LIN {X 0,Y 573.243,Z 369.081,A -85,B 0,C 180,E1 -2301.298,E2 -2301.298} C_VEL
LIN {X 0,Y 573.218,Z 369.085,A -85,B 0,C 180,E1 -2304.019,E2 -2304.019} C_VEL
LIN {X 0,Y 573.243,Z 369.081,A -85,B 0,C 180,E1 -2306.516,E2 -2306.516} C_VEL
LIN {X 0,Y 573.233,Z 369.084,A -85,B 0,C 180,E1 -2309.118,E2 -2309.118} C_VEL
LIN {X 0,Y 573.24,Z 369.081,A -85,B 0,C 180,E1 -2311.435,E2 -2311.435} C_VEL
LIN {X 0,Y 573.267,Z 369.078,A -85,B 0,C 180,E1 -2313.81,E2 -2313.81} C_VEL
LIN {X 0,Y 573.232,Z 369.084,A -85,B 0,C 180,E1 -2316.134,E2 -2316.134} C_VEL
LIN {X 0,Y 573.254,Z 369.081,A -85,B 0,C 180,E1 -2319.174,E2 -2319.174} C_VEL
LIN {X 0,Y 573.232,Z 369.084,A -85,B 0,C 180,E1 -2321.411,E2 -2321.411} C_VEL
LIN {X 0,Y 573.253,Z 369.082,A -85,B 0,C 180,E1 -2323.622,E2 -2323.622} C_VEL
LIN {X 0,Y 573.276,Z 369.078,A -85,B 0,C 180,E1 -2325.807,E2 -2325.807} C_VEL
LIN {X 0,Y 573.267,Z 369.08,A -85,B 0,C 180,E1 -2328.745,E2 -2328.745} C_VEL
LIN {X 0,Y 573.292,Z 369.075,A -85,B 0,C 180,E1 -2331.541,E2 -2331.541} C_VEL
LIN {X 0,Y 573.291,Z 369.075,A -85,B 0,C 180,E1 -2334.372,E2 -2334.372} C_VEL
LIN {X 0,Y 573.314,Z 369.074,A -85,B 0,C 180,E1 -2337.892,E2 -2337.892} C_VEL
LIN {X 0,Y 573.331,Z 369.07,A -85,B 0,C 180,E1 -2340.702,E2 -2340.702} C_VEL
LIN {X 0,Y 573.238,Z 369.082,A -85,B 0,C 180,E1 -2343.514,E2 -2343.514} C_VEL
LIN {X 0,Y 573.294,Z 369.075,A -85,B 0,C 180,E1 -2345.628,E2 -2345.628} C_VEL
LIN {X 0,Y 573.292,Z 369.076,A -85,B 0,C 180,E1 -2348.459,E2 -2348.459} C_VEL
LIN {X 0,Y 573.275,Z 369.078,A -85,B 0,C 180,E1 -2351.312,E2 -2351.312} C_VEL
LIN {X 0,Y 573.284,Z 369.078,A -85,B 0,C 180,E1 -2354.424,E2 -2354.424} C_VEL
LIN {X 0,Y 573.262,Z 369.079,A -85,B 0,C 180,E1 -2357.111,E2 -2357.111} C_VEL
LIN {X 0,Y 573.244,Z 369.081,A -85,B 0,C 180,E1 -2360.077,E2 -2360.077} C_VEL
LIN {X 0,Y 573.237,Z 369.082,A -85,B 0,C 180,E1 -2362.338,E2 -2362.338} C_VEL
LIN {X 0,Y 573.254,Z 369.079,A -85,B 0,C 180,E1 -2364.39,E2 -2364.39} C_VEL
LIN {X 0,Y 572.627,Z 369.16,A -85,B 0,C 180,E1 -2364.976,E2 -2364.976} C_VEL
LIN {X 0,Y 569.784,Z 369.514,A -85,B 0,C 180,E1 -2365.927,E2 -2365.927} C_VEL
LIN {X 0,Y 567.352,Z 369.817,A -85,B 0,C 180,E1 -2366.693,E2 -2366.693} C_VEL
LIN {X 0,Y 566.297,Z 369.948,A -85,B 0,C 180,E1 -2367.284,E2 -2367.284} C_VEL
LIN {X 0,Y 566.207,Z 369.957,A -85,B 0,C 180,E1 -2367.484,E2 -2367.484} C_VEL
LIN {X 0,Y 566.205,Z 369.958,A -85,B 0,C 180,E1 -2369.769,E2 -2369.769} C_VEL
LIN {X 0,Y 566.208,Z 369.958,A -85,B 0,C 180,E1 -2372.43,E2 -2372.43} C_VEL
LIN {X 0,Y 566.184,Z 369.961,A -85,B 0,C 180,E1 -2374.989,E2 -2374.989} C_VEL
LIN {X 0,Y 566.2,Z 369.961,A -85,B 0,C 180,E1 -2377.461,E2 -2377.461} C_VEL
LIN {X 0,Y 566.211,Z 369.957,A -85,B 0,C 180,E1 -2380.199,E2 -2380.199} C_VEL
LIN {X 0,Y 566.204,Z 369.958,A -85,B 0,C 180,E1 -2383.054,E2 -2383.054} C_VEL
LIN {X 0,Y 566.198,Z 369.958,A -85,B 0,C 180,E1 -2386.049,E2 -2386.049} C_VEL
LIN {X 0,Y 566.185,Z 369.963,A -85,B 0,C 180,E1 -2388.861,E2 -2388.861} C_VEL
LIN {X 0,Y 566.218,Z 369.956,A -85,B 0,C 180,E1 -2391.441,E2 -2391.441} C_VEL
LIN {X 0,Y 566.168,Z 369.963,A -85,B 0,C 180,E1 -2394.307,E2 -2394.307} C_VEL
LIN {X 0,Y 566.225,Z 369.957,A -85,B 0,C 180,E1 -2396.897,E2 -2396.897} C_VEL
LIN {X 0,Y 566.181,Z 369.961,A -85,B 0,C 180,E1 -2399.406,E2 -2399.406} C_VEL
LIN {X 0,Y 566.2,Z 369.958,A -85,B 0,C 180,E1 -2401.856,E2 -2401.856} C_VEL
LIN {X 0,Y 566.219,Z 369.957,A -85,B 0,C 180,E1 -2404.25,E2 -2404.25} C_VEL
LIN {X 0,Y 566.178,Z 369.962,A -85,B 0,C 180,E1 -2406.718,E2 -2406.718} C_VEL
LIN {X 0,Y 566.219,Z 369.957,A -85,B 0,C 180,E1 -2409.662,E2 -2409.662} C_VEL
LIN {X 0,Y 566.205,Z 369.96,A -85,B 0,C 180,E1 -2412.667,E2 -2412.667} C_VEL
LIN {X 0,Y 566.24,Z 369.955,A -85,B 0,C 180,E1 -2415.626,E2 -2415.626} C_VEL
LIN {X 0,Y 566.111,Z 369.972,A -85,B 0,C 180,E1 -2418.542,E2 -2418.542} C_VEL
LIN {X 0,Y 566.05,Z 370.2,A -85,B 0,C 180,E1 -2419.266,E2 -2419.266} C_VEL
LIN {X 0,Y 566.031,Z 373.545,A -85,B 0,C 180,E1 -2422.149,E2 -2422.149} C_VEL
LIN {X 0,Y 566.036,Z 376.76,A -85,B 0,C 180,E1 -2425.013,E2 -2425.013} C_VEL
LIN {X 0,Y 565.932,Z 379.928,A -85,B 0,C 180,E1 -2427.864,E2 -2427.864} C_VEL
LIN {X 0,Y 565.858,Z 383.215,A -85,B 0,C 180,E1 -2430.71,E2 -2430.71} C_VEL
LIN {X 0,Y 565.899,Z 386.764,A -85,B 0,C 180,E1 -2433.559,E2 -2433.559} C_VEL
LIN {X 0,Y 565.875,Z 390.539,A -85,B 0,C 180,E1 -2436.497,E2 -2436.497} C_VEL
LIN {X 0,Y 565.805,Z 394.183,A -85,B 0,C 180,E1 -2439.291,E2 -2439.291} C_VEL
LIN {X 0,Y 565.863,Z 395.844,A -85,B 0,C 180,E1 -2440.441,E2 -2440.441} C_VEL
LIN {X 0,Y 566.862,Z 403.182,A -85,B 0,C 180,E1 -2440.626,E2 -2440.626} C_VEL
LIN {X 0,Y 566.816,Z 416.303,A -85,B 0,C 180,E1 -2441.032,E2 -2441.032} C_VEL
LIN {X 0,Y 566.624,Z 427.611,A -85,B 0,C 180,E1 -2441.518,E2 -2441.518} C_VEL
LIN {X 0,Y 566.478,Z 439.306,A -85,B 0,C 180,E1 -2442.174,E2 -2442.174} C_VEL
LIN {X 0,Y 566.351,Z 450.857,A -85,B 0,C 180,E1 -2442.996,E2 -2442.996} C_VEL
LIN {X 0,Y 566.205,Z 460.179,A -85,B 0,C 180,E1 -2443.822,E2 -2443.822} C_VEL
LIN {X 0,Y 566.12,Z 468.385,A -85,B 0,C 180,E1 -2444.705,E2 -2444.705} C_VEL
LIN {X 0,Y 566.031,Z 477.042,A -85,B 0,C 180,E1 -2445.851,E2 -2445.851} C_VEL
LIN {X 0,Y 565.988,Z 484.113,A -85,B 0,C 180,E1 -2447.035,E2 -2447.035} C_VEL
LIN {X 0,Y 565.927,Z 489.058,A -85,B 0,C 180,E1 -2448.085,E2 -2448.085} C_VEL
LIN {X 0,Y 565.888,Z 493.37,A -85,B 0,C 180,E1 -2449.287,E2 -2449.287} C_VEL
LIN {X 0,Y 565.86,Z 496.126,A -85,B 0,C 180,E1 -2450.349,E2 -2450.349} C_VEL
LIN {X 0,Y 565.859,Z 497.849,A -85,B 0,C 180,E1 -2451.329,E2 -2451.329} C_VEL
LIN {X 0,Y 565.839,Z 498.918,A -85,B 0,C 180,E1 -2452.644,E2 -2452.644} C_VEL
LIN {X 0,Y 565.845,Z 498.924,A -85,B 0,C 180,E1 -2453.417,E2 -2453.417} C_VEL
LIN {X 0,Y 565.826,Z 498.482,A -85,B 0,C 180,E1 -2454.196,E2 -2454.196} C_VEL
LIN {X 0,Y 565.847,Z 497.517,A -85,B 0,C 180,E1 -2454.977,E2 -2454.977} C_VEL
LIN {X 0,Y 565.853,Z 496.078,A -85,B 0,C 180,E1 -2455.765,E2 -2455.765} C_VEL
LIN {X 0,Y 565.901,Z 492.922,A -85,B 0,C 180,E1 -2456.953,E2 -2456.953} C_VEL
LIN {X 0,Y 565.923,Z 488.418,A -85,B 0,C 180,E1 -2458.156,E2 -2458.156} C_VEL
LIN {X 0,Y 565.975,Z 482.771,A -85,B 0,C 180,E1 -2459.301,E2 -2459.301} C_VEL
LIN {X 0,Y 566.088,Z 476.006,A -85,B 0,C 180,E1 -2460.39,E2 -2460.39} C_VEL
LIN {X 0,Y 566.15,Z 468.073,A -85,B 0,C 180,E1 -2461.422,E2 -2461.422} C_VEL
LIN {X 0,Y 566.279,Z 458.336,A -85,B 0,C 180,E1 -2462.442,E2 -2462.442} C_VEL
LIN {X 0,Y 566.385,Z 448.167,A -85,B 0,C 180,E1 -2463.301,E2 -2463.301} C_VEL
LIN {X 0,Y 566.54,Z 437.358,A -85,B 0,C 180,E1 -2464.038,E2 -2464.038} C_VEL
LIN {X 0,Y 566.692,Z 425.446,A -85,B 0,C 180,E1 -2464.673,E2 -2464.673} C_VEL
LIN {X 0,Y 566.777,Z 412.677,A -85,B 0,C 180,E1 -2465.186,E2 -2465.186} C_VEL
LIN {X 0,Y 566.713,Z 400.738,A -85,B 0,C 180,E1 -2465.528,E2 -2465.528} C_VEL
LIN {X 0,Y 565.86,Z 395.663,A -85,B 0,C 180,E1 -2465.673,E2 -2465.673} C_VEL
LIN {X 0,Y 565.839,Z 391.945,A -85,B 0,C 180,E1 -2468.511,E2 -2468.511} C_VEL
LIN {X 0,Y 565.879,Z 388.515,A -85,B 0,C 180,E1 -2471.163,E2 -2471.163} C_VEL
LIN {X 0,Y 565.888,Z 384.824,A -85,B 0,C 180,E1 -2474.063,E2 -2474.063} C_VEL
LIN {X 0,Y 565.914,Z 382.456,A -85,B 0,C 180,E1 -2476.075,E2 -2476.075} C_VEL
LIN {X 0,Y 565.949,Z 379.413,A -85,B 0,C 180,E1 -2478.84,E2 -2478.84} C_VEL
LIN {X 0,Y 565.95,Z 376.333,A -85,B 0,C 180,E1 -2481.618,E2 -2481.618} C_VEL
LIN {X 0,Y 566.006,Z 373.303,A -85,B 0,C 180,E1 -2484.296,E2 -2484.296} C_VEL
LIN {X 0,Y 566.029,Z 370.291,A -85,B 0,C 180,E1 -2486.885,E2 -2486.885} C_VEL
LIN {X 0,Y 566.128,Z 369.968,A -85,B 0,C 180,E1 -2488.574,E2 -2488.574} C_VEL
LIN {X 0,Y 566.181,Z 369.963,A -85,B 0,C 180,E1 -2491.046,E2 -2491.046} C_VEL
LIN {X 0,Y 566.229,Z 369.955,A -85,B 0,C 180,E1 -2493.46,E2 -2493.46} C_VEL
LIN {X 0,Y 566.198,Z 369.957,A -85,B 0,C 180,E1 -2495.819,E2 -2495.819} C_VEL
LIN {X 0,Y 566.196,Z 369.957,A -85,B 0,C 180,E1 -2498.576,E2 -2498.576} C_VEL
LIN {X 0,Y 566.202,Z 369.956,A -85,B 0,C 180,E1 -2501.172,E2 -2501.172} C_VEL
LIN {X 0,Y 566.19,Z 369.958,A -85,B 0,C 180,E1 -2504.152,E2 -2504.152} C_VEL
LIN {X 0,Y 566.186,Z 369.958,A -85,B 0,C 180,E1 -2506.359,E2 -2506.359} C_VEL
LIN {X 0,Y 566.235,Z 369.952,A -85,B 0,C 180,E1 -2509.27,E2 -2509.27} C_VEL
LIN {X 0,Y 566.226,Z 369.954,A -85,B 0,C 180,E1 -2512.153,E2 -2512.153} C_VEL
LIN {X 0,Y 566.274,Z 369.949,A -85,B 0,C 180,E1 -2515.016,E2 -2515.016} C_VEL
LIN {X 0,Y 566.275,Z 369.95,A -85,B 0,C 180,E1 -2517.866,E2 -2517.866} C_VEL
LIN {X 0,Y 566.293,Z 369.949,A -85,B 0,C 180,E1 -2520.711,E2 -2520.711} C_VEL
LIN {X 0,Y 566.264,Z 369.948,A -85,B 0,C 180,E1 -2522.846,E2 -2522.846} C_VEL
LIN {X 0,Y 566.244,Z 369.951,A -85,B 0,C 180,E1 -2525.699,E2 -2525.699} C_VEL
LIN {X 0,Y 566.214,Z 369.956,A -85,B 0,C 180,E1 -2528.566,E2 -2528.566} C_VEL
LIN {X 0,Y 566.23,Z 369.956,A -85,B 0,C 180,E1 -2531.455,E2 -2531.455} C_VEL
LIN {X 0,Y 566.213,Z 369.957,A -85,B 0,C 180,E1 -2534.508,E2 -2534.508} C_VEL
LIN {X 0,Y 566.186,Z 369.96,A -85,B 0,C 180,E1 -2537.332,E2 -2537.332} C_VEL
LIN {X 0,Y 566.197,Z 369.96,A -85,B 0,C 180,E1 -2539.581,E2 -2539.581} C_VEL
LIN {X 0,Y 566.207,Z 369.958,A -85,B 0,C 180,E1 -2542.631,E2 -2542.631} C_VEL
LIN {X 0,Y 566.198,Z 369.961,A -85,B 0,C 180,E1 -2545.031,E2 -2545.031} C_VEL
LIN {X 0,Y 566.209,Z 369.957,A -85,B 0,C 180,E1 -2547.339,E2 -2547.339} C_VEL
LIN {X 0,Y 566.185,Z 369.959,A -85,B 0,C 180,E1 -2549.77,E2 -2549.77} C_VEL
LIN {X 0,Y 566.194,Z 369.958,A -85,B 0,C 180,E1 -2552.433,E2 -2552.433} C_VEL
LIN {X 0,Y 566.198,Z 369.958,A -85,B 0,C 180,E1 -2554.996,E2 -2554.996} C_VEL
LIN {X 0,Y 566.182,Z 369.962,A -85,B 0,C 180,E1 -2557.462,E2 -2557.462} C_VEL
LIN {X 0,Y 566.211,Z 369.958,A -85,B 0,C 180,E1 -2560.199,E2 -2560.199} C_VEL
LIN {X 0,Y 566.188,Z 369.961,A -85,B 0,C 180,E1 -2563.056,E2 -2563.056} C_VEL
LIN {X 0,Y 566.19,Z 369.96,A -85,B 0,C 180,E1 -2566.05,E2 -2566.05} C_VEL
LIN {X 0,Y 566.21,Z 369.957,A -85,B 0,C 180,E1 -2568.866,E2 -2568.866} C_VEL
LIN {X 0,Y 566.18,Z 369.961,A -85,B 0,C 180,E1 -2571.639,E2 -2571.639} C_VEL
LIN {X 0,Y 566.233,Z 370.124,A -85,B 0,C 180,E1 -2573.047,E2 -2573.047} C_VEL
LIN {X 0,Y 566.84,Z 373.924,A -85,B 0,C 180,E1 -2574.36,E2 -2574.36} C_VEL
LIN {X 0,Y 566.738,Z 381.867,A -85,B 0,C 180,E1 -2576.934,E2 -2576.934} C_VEL
LIN {X 0,Y 566.604,Z 389.811,A -85,B 0,C 180,E1 -2579.435,E2 -2579.435} C_VEL
LIN {X 0,Y 566.501,Z 399.078,A -85,B 0,C 180,E1 -2582.277,E2 -2582.277} C_VEL
LIN {X 0,Y 566.407,Z 408.345,A -85,B 0,C 180,E1 -2585.049,E2 -2585.049} C_VEL
LIN {X 0,Y 566.319,Z 418.936,A -85,B 0,C 180,E1 -2588.144,E2 -2588.144} C_VEL
LIN {X 0,Y 566.19,Z 429.527,A -85,B 0,C 180,E1 -2591.174,E2 -2591.174} C_VEL
LIN {X 0,Y 566.114,Z 440.118,A -85,B 0,C 180,E1 -2594.152,E2 -2594.152} C_VEL
LIN {X 0,Y 566.022,Z 449.385,A -85,B 0,C 180,E1 -2596.722,E2 -2596.722} C_VEL
LIN {X 0,Y 566.013,Z 451.536,A -85,B 0,C 180,E1 -2597.315,E2 -2597.315} C_VEL
LIN {X 0,Y 566.93,Z 458.454,A -85,B 0,C 180,E1 -2597.472,E2 -2597.472} C_VEL
LIN {X 0,Y 566.856,Z 470.552,A -85,B 0,C 180,E1 -2597.789,E2 -2597.789} C_VEL
LIN {X 0,Y 566.69,Z 482.355,A -85,B 0,C 180,E1 -2598.23,E2 -2598.23} C_VEL
LIN {X 0,Y 566.541,Z 494.944,A -85,B 0,C 180,E1 -2598.866,E2 -2598.866} C_VEL
LIN {X 0,Y 566.432,Z 505.501,A -85,B 0,C 180,E1 -2599.547,E2 -2599.547} C_VEL
LIN {X 0,Y 566.3,Z 515.665,A -85,B 0,C 180,E1 -2600.357,E2 -2600.357} C_VEL
LIN {X 0,Y 566.165,Z 524.801,A -85,B 0,C 180,E1 -2601.255,E2 -2601.255} C_VEL
LIN {X 0,Y 566.079,Z 533.702,A -85,B 0,C 180,E1 -2602.332,E2 -2602.332} C_VEL
LIN {X 0,Y 565.966,Z 540.964,A -85,B 0,C 180,E1 -2603.424,E2 -2603.424} C_VEL
LIN {X 0,Y 566.003,Z 545.688,A -85,B 0,C 180,E1 -2604.301,E2 -2604.301} C_VEL
LIN {X 0,Y 565.933,Z 550.377,A -85,B 0,C 180,E1 -2605.372,E2 -2605.372} C_VEL
LIN {X 0,Y 565.926,Z 553.961,A -85,B 0,C 180,E1 -2606.441,E2 -2606.441} C_VEL
LIN {X 0,Y 565.877,Z 555.812,A -85,B 0,C 180,E1 -2607.154,E2 -2607.154} C_VEL
LIN {X 0,Y 565.84,Z 557.202,A -85,B 0,C 180,E1 -2607.866,E2 -2607.866} C_VEL
LIN {X 0,Y 565.841,Z 558.785,A -85,B 0,C 180,E1 -2609.29,E2 -2609.29} C_VEL
LIN {X 0,Y 565.839,Z 559,A -85,B 0,C 180,E1 -2610.001,E2 -2610.001} C_VEL
LIN {X 0,Y 565.846,Z 558.184,A -85,B 0,C 180,E1 -2611.425,E2 -2611.425} C_VEL
LIN {X 0,Y 565.841,Z 557.199,A -85,B 0,C 180,E1 -2612.137,E2 -2612.137} C_VEL
LIN {X 0,Y 565.878,Z 555.807,A -85,B 0,C 180,E1 -2612.849,E2 -2612.849} C_VEL
LIN {X 0,Y 565.927,Z 552.892,A -85,B 0,C 180,E1 -2613.918,E2 -2613.918} C_VEL
LIN {X 0,Y 565.878,Z 548.944,A -85,B 0,C 180,E1 -2614.989,E2 -2614.989} C_VEL
LIN {X 0,Y 566.002,Z 543.86,A -85,B 0,C 180,E1 -2616.06,E2 -2616.06} C_VEL
LIN {X 0,Y 566.042,Z 537.461,A -85,B 0,C 180,E1 -2617.134,E2 -2617.134} C_VEL
LIN {X 0,Y 566.134,Z 529.468,A -85,B 0,C 180,E1 -2618.209,E2 -2618.209} C_VEL
LIN {X 0,Y 566.23,Z 521.325,A -85,B 0,C 180,E1 -2619.107,E2 -2619.107} C_VEL
LIN {X 0,Y 566.347,Z 511.388,A -85,B 0,C 180,E1 -2620.006,E2 -2620.006} C_VEL
LIN {X 0,Y 566.52,Z 500.298,A -85,B 0,C 180,E1 -2620.807,E2 -2620.807} C_VEL
LIN {X 0,Y 566.611,Z 487.929,A -85,B 0,C 180,E1 -2621.511,E2 -2621.511} C_VEL
LIN {X 0,Y 566.778,Z 475.734,A -85,B 0,C 180,E1 -2622.034,E2 -2622.034} C_VEL
LIN {X 0,Y 566.928,Z 462.304,A -85,B 0,C 180,E1 -2622.44,E2 -2622.44} C_VEL
LIN {X 0,Y 566.631,Z 455.461,A -85,B 0,C 180,E1 -2622.594,E2 -2622.594} C_VEL
LIN {X 0,Y 566.015,Z 451.526,A -85,B 0,C 180,E1 -2622.688,E2 -2622.688} C_VEL
LIN {X 0,Y 566.09,Z 441.432,A -85,B 0,C 180,E1 -2625.482,E2 -2625.482} C_VEL
LIN {X 0,Y 566.176,Z 430.841,A -85,B 0,C 180,E1 -2628.454,E2 -2628.454} C_VEL
LIN {X 0,Y 566.242,Z 421.573,A -85,B 0,C 180,E1 -2631.097,E2 -2631.097} C_VEL
LIN {X 0,Y 566.344,Z 412.306,A -85,B 0,C 180,E1 -2633.786,E2 -2633.786} C_VEL
LIN {X 0,Y 566.482,Z 403.039,A -85,B 0,C 180,E1 -2636.529,E2 -2636.529} C_VEL
LIN {X 0,Y 566.54,Z 393.772,A -85,B 0,C 180,E1 -2639.342,E2 -2639.342} C_VEL
LIN {X 0,Y 566.756,Z 384.505,A -85,B 0,C 180,E1 -2642.224,E2 -2642.224} C_VEL
LIN {X 0,Y 566.841,Z 376.562,A -85,B 0,C 180,E1 -2644.774,E2 -2644.774} C_VEL
LIN {X 0,Y 566.583,Z 372.063,A -85,B 0,C 180,E1 -2646.266,E2 -2646.266} C_VEL
LIN {X 0,Y 566.24,Z 369.954,A -85,B 0,C 180,E1 -2647.012,E2 -2647.012} C_VEL
LIN {X 0,Y 566.219,Z 369.957,A -85,B 0,C 180,E1 -2649.686,E2 -2649.686} C_VEL
LIN {X 0,Y 566.206,Z 369.958,A -85,B 0,C 180,E1 -2652.917,E2 -2652.917} C_VEL
LIN {X 0,Y 566.199,Z 369.959,A -85,B 0,C 180,E1 -2656.05,E2 -2656.05} C_VEL
LIN {X 0,Y 566.209,Z 369.958,A -85,B 0,C 180,E1 -2659.215,E2 -2659.215} C_VEL
LIN {X 0,Y 566.188,Z 369.962,A -85,B 0,C 180,E1 -2661.637,E2 -2661.637} C_VEL
LIN {X 0,Y 566.167,Z 369.963,A -85,B 0,C 180,E1 -2664.308,E2 -2664.308} C_VEL
LIN {X 0,Y 566.208,Z 369.96,A -85,B 0,C 180,E1 -2666.897,E2 -2666.897} C_VEL
LIN {X 0,Y 566.185,Z 369.96,A -85,B 0,C 180,E1 -2669.407,E2 -2669.407} C_VEL
LIN {X 0,Y 566.199,Z 369.959,A -85,B 0,C 180,E1 -2671.857,E2 -2671.857} C_VEL
LIN {X 0,Y 566.217,Z 369.959,A -85,B 0,C 180,E1 -2674.251,E2 -2674.251} C_VEL
LIN {X 0,Y 566.176,Z 369.962,A -85,B 0,C 180,E1 -2676.719,E2 -2676.719} C_VEL
LIN {X 0,Y 566.217,Z 369.957,A -85,B 0,C 180,E1 -2679.663,E2 -2679.663} C_VEL
LIN {X 0,Y 566.204,Z 369.959,A -85,B 0,C 180,E1 -2682.668,E2 -2682.668} C_VEL
LIN {X 0,Y 566.237,Z 369.956,A -85,B 0,C 180,E1 -2685.627,E2 -2685.627} C_VEL
LIN {X 0,Y 566.239,Z 369.956,A -85,B 0,C 180,E1 -2688.675,E2 -2688.675} C_VEL
LIN {X 0,Y 566.236,Z 369.953,A -85,B 0,C 180,E1 -2691.434,E2 -2691.434} C_VEL
LIN {X 0,Y 566.26,Z 369.951,A -85,B 0,C 180,E1 -2694.302,E2 -2694.302} C_VEL
LIN {X 0,Y 566.285,Z 369.949,A -85,B 0,C 180,E1 -2697.866,E2 -2697.866} C_VEL
LIN {X 0,Y 566.302,Z 369.946,A -85,B 0,C 180,E1 -2700.711,E2 -2700.711} C_VEL
LIN {X 0,Y 566.275,Z 369.949,A -85,B 0,C 180,E1 -2702.845,E2 -2702.845} C_VEL
LIN {X 0,Y 566.262,Z 369.951,A -85,B 0,C 180,E1 -2705.698,E2 -2705.698} C_VEL
LIN {X 0,Y 566.236,Z 369.954,A -85,B 0,C 180,E1 -2708.566,E2 -2708.566} C_VEL
LIN {X 0,Y 566.246,Z 369.955,A -85,B 0,C 180,E1 -2711.454,E2 -2711.454} C_VEL
LIN {X 0,Y 566.237,Z 369.956,A -85,B 0,C 180,E1 -2714.506,E2 -2714.506} C_VEL
LIN {X 0,Y 566.202,Z 369.958,A -85,B 0,C 180,E1 -2717.332,E2 -2717.332} C_VEL
LIN {X 0,Y 566.21,Z 369.957,A -85,B 0,C 180,E1 -2720.337,E2 -2720.337} C_VEL
LIN {X 0,Y 566.177,Z 369.962,A -85,B 0,C 180,E1 -2723.282,E2 -2723.282} C_VEL
LIN {X 0,Y 566.213,Z 369.958,A -85,B 0,C 180,E1 -2725.749,E2 -2725.749} C_VEL
LIN {X 0,Y 566.207,Z 369.957,A -85,B 0,C 180,E1 -2727.484,E2 -2727.484} C_VEL
LIN {X 0,Y 565.527,Z 370.044,A -85,B 0,C 180,E1 -2728.078,E2 -2728.078} C_VEL
LIN {X 0,Y 562.661,Z 370.401,A -85,B 0,C 180,E1 -2729.042,E2 -2729.042} C_VEL
LIN {X 0,Y 560.251,Z 370.7,A -85,B 0,C 180,E1 -2729.817,E2 -2729.817} C_VEL
LIN {X 0,Y 559.224,Z 370.828,A -85,B 0,C 180,E1 -2730.416,E2 -2730.416} C_VEL
LIN {X 0,Y 559.144,Z 370.837,A -85,B 0,C 180,E1 -2730.619,E2 -2730.619} C_VEL
LIN {X 0,Y 559.163,Z 370.836,A -85,B 0,C 180,E1 -2733.575,E2 -2733.575} C_VEL
LIN {X 0,Y 559.15,Z 370.838,A -85,B 0,C 180,E1 -2736.445,E2 -2736.445} C_VEL
LIN {X 0,Y 559.176,Z 370.833,A -85,B 0,C 180,E1 -2738.934,E2 -2738.934} C_VEL
LIN {X 0,Y 559.166,Z 370.835,A -85,B 0,C 180,E1 -2741.77,E2 -2741.77} C_VEL
LIN {X 0,Y 559.136,Z 370.84,A -85,B 0,C 180,E1 -2744.74,E2 -2744.74} C_VEL
LIN {X 0,Y 559.179,Z 370.834,A -85,B 0,C 180,E1 -2747.863,E2 -2747.863} C_VEL
LIN {X 0,Y 559.182,Z 370.834,A -85,B 0,C 180,E1 -2751.066,E2 -2751.066} C_VEL
LIN {X 0,Y 559.145,Z 370.839,A -85,B 0,C 180,E1 -2753.789,E2 -2753.789} C_VEL
LIN {X 0,Y 559.168,Z 370.835,A -85,B 0,C 180,E1 -2756.425,E2 -2756.425} C_VEL
LIN {X 0,Y 559.158,Z 370.837,A -85,B 0,C 180,E1 -2758.98,E2 -2758.98} C_VEL
LIN {X 0,Y 559.174,Z 370.833,A -85,B 0,C 180,E1 -2761.618,E2 -2761.618} C_VEL
LIN {X 0,Y 559.185,Z 370.831,A -85,B 0,C 180,E1 -2763.902,E2 -2763.902} C_VEL
LIN {X 0,Y 559.147,Z 370.839,A -85,B 0,C 180,E1 -2766.57,E2 -2766.57} C_VEL
LIN {X 0,Y 559.185,Z 370.834,A -85,B 0,C 180,E1 -2769.395,E2 -2769.395} C_VEL
LIN {X 0,Y 559.148,Z 370.838,A -85,B 0,C 180,E1 -2771.685,E2 -2771.685} C_VEL
LIN {X 0,Y 559.169,Z 370.835,A -85,B 0,C 180,E1 -2773.947,E2 -2773.947} C_VEL
LIN {X 0,Y 559.179,Z 370.833,A -85,B 0,C 180,E1 -2776.183,E2 -2776.183} C_VEL
LIN {X 0,Y 559.086,Z 370.847,A -85,B 0,C 180,E1 -2778.667,E2 -2778.667} C_VEL
LIN {X 0,Y 558.996,Z 370.858,A -85,B 0,C 180,E1 -2779.128,E2 -2779.128} C_VEL
LIN {X 0,Y 558.961,Z 374.055,A -85,B 0,C 180,E1 -2782.049,E2 -2782.049} C_VEL
LIN {X 0,Y 558.985,Z 377.336,A -85,B 0,C 180,E1 -2784.95,E2 -2784.95} C_VEL
LIN {X 0,Y 558.859,Z 380.549,A -85,B 0,C 180,E1 -2787.837,E2 -2787.837} C_VEL
LIN {X 0,Y 558.88,Z 382.996,A -85,B 0,C 180,E1 -2789.999,E2 -2789.999} C_VEL
LIN {X 0,Y 558.762,Z 386.292,A -85,B 0,C 180,E1 -2792.882,E2 -2792.882} C_VEL
LIN {X 0,Y 558.822,Z 389.89,A -85,B 0,C 180,E1 -2795.773,E2 -2795.773} C_VEL
LIN {X 0,Y 558.755,Z 393.622,A -85,B 0,C 180,E1 -2798.68,E2 -2798.68} C_VEL
LIN {X 0,Y 558.758,Z 395.823,A -85,B 0,C 180,E1 -2800.278,E2 -2800.278} C_VEL
LIN {X 0,Y 559.933,Z 403.771,A -85,B 0,C 180,E1 -2800.484,E2 -2800.484} C_VEL
LIN {X 0,Y 559.87,Z 416.607,A -85,B 0,C 180,E1 -2800.893,E2 -2800.893} C_VEL
LIN {X 0,Y 559.641,Z 428.895,A -85,B 0,C 180,E1 -2801.439,E2 -2801.439} C_VEL
LIN {X 0,Y 559.462,Z 440.992,A -85,B 0,C 180,E1 -2802.145,E2 -2802.145} C_VEL
LIN {X 0,Y 559.323,Z 451.065,A -85,B 0,C 180,E1 -2802.885,E2 -2802.885} C_VEL
LIN {X 0,Y 559.161,Z 461.247,A -85,B 0,C 180,E1 -2803.814,E2 -2803.814} C_VEL
LIN {X 0,Y 559.049,Z 469.59,A -85,B 0,C 180,E1 -2804.746,E2 -2804.746} C_VEL
LIN {X 0,Y 558.956,Z 477.784,A -85,B 0,C 180,E1 -2805.869,E2 -2805.869} C_VEL
LIN {X 0,Y 558.923,Z 483.323,A -85,B 0,C 180,E1 -2806.809,E2 -2806.809} C_VEL
LIN {X 0,Y 558.836,Z 488.743,A -85,B 0,C 180,E1 -2807.944,E2 -2807.944} C_VEL
LIN {X 0,Y 558.81,Z 492.914,A -85,B 0,C 180,E1 -2809.085,E2 -2809.085} C_VEL
LIN {X 0,Y 558.76,Z 495.051,A -85,B 0,C 180,E1 -2809.851,E2 -2809.851} C_VEL
LIN {X 0,Y 558.759,Z 496.735,A -85,B 0,C 180,E1 -2810.619,E2 -2810.619} C_VEL
LIN {X 0,Y 558.764,Z 498.012,A -85,B 0,C 180,E1 -2811.447,E2 -2811.447} C_VEL
LIN {X 0,Y 558.737,Z 498.683,A -85,B 0,C 180,E1 -2812.168,E2 -2812.168} C_VEL
LIN {X 0,Y 558.755,Z 498.943,A -85,B 0,C 180,E1 -2813.337,E2 -2813.337} C_VEL
LIN {X 0,Y 558.757,Z 498.145,A -85,B 0,C 180,E1 -2814.522,E2 -2814.522} C_VEL
LIN {X 0,Y 558.751,Z 497.025,A -85,B 0,C 180,E1 -2815.317,E2 -2815.317} C_VEL
LIN {X 0,Y 558.813,Z 493.652,A -85,B 0,C 180,E1 -2816.754,E2 -2816.754} C_VEL
LIN {X 0,Y 558.838,Z 489.228,A -85,B 0,C 180,E1 -2818.025,E2 -2818.025} C_VEL
LIN {X 0,Y 558.909,Z 482.859,A -85,B 0,C 180,E1 -2819.365,E2 -2819.365} C_VEL
LIN {X 0,Y 559.016,Z 475.168,A -85,B 0,C 180,E1 -2820.606,E2 -2820.606} C_VEL
LIN {X 0,Y 559.102,Z 466.635,A -85,B 0,C 180,E1 -2821.696,E2 -2821.696} C_VEL
LIN {X 0,Y 559.273,Z 456.793,A -85,B 0,C 180,E1 -2822.705,E2 -2822.705} C_VEL
LIN {X 0,Y 559.433,Z 446.565,A -85,B 0,C 180,E1 -2823.554,E2 -2823.554} C_VEL
LIN {X 0,Y 559.57,Z 435.653,A -85,B 0,C 180,E1 -2824.278,E2 -2824.278} C_VEL
LIN {X 0,Y 559.759,Z 423.899,A -85,B 0,C 180,E1 -2824.891,E2 -2824.891} C_VEL
LIN {X 0,Y 559.885,Z 410.658,A -85,B 0,C 180,E1 -2825.407,E2 -2825.407} C_VEL
LIN {X 0,Y 559.735,Z 401.403,A -85,B 0,C 180,E1 -2825.67,E2 -2825.67} C_VEL
LIN {X 0,Y 558.754,Z 395.676,A -85,B 0,C 180,E1 -2825.826,E2 -2825.826} C_VEL
LIN {X 0,Y 558.742,Z 391.618,A -85,B 0,C 180,E1 -2828.967,E2 -2828.967} C_VEL
LIN {X 0,Y 558.789,Z 388.008,A -85,B 0,C 180,E1 -2831.802,E2 -2831.802} C_VEL
LIN {X 0,Y 558.857,Z 384.581,A -85,B 0,C 180,E1 -2834.765,E2 -2834.765} C_VEL
LIN {X 0,Y 558.858,Z 381.052,A -85,B 0,C 180,E1 -2837.895,E2 -2837.895} C_VEL
LIN {X 0,Y 558.885,Z 378.677,A -85,B 0,C 180,E1 -2840.109,E2 -2840.109} C_VEL
LIN {X 0,Y 558.917,Z 375.56,A -85,B 0,C 180,E1 -2842.874,E2 -2842.874} C_VEL
LIN {X 0,Y 558.945,Z 372.481,A -85,B 0,C 180,E1 -2845.541,E2 -2845.541} C_VEL
LIN {X 0,Y 559.003,Z 370.858,A -85,B 0,C 180,E1 -2847.385,E2 -2847.385} C_VEL
LIN {X 0,Y 559.171,Z 370.833,A -85,B 0,C 180,E1 -2850.134,E2 -2850.134} C_VEL
LIN {X 0,Y 559.165,Z 370.833,A -85,B 0,C 180,E1 -2853.169,E2 -2853.169} C_VEL
LIN {X 0,Y 559.148,Z 370.836,A -85,B 0,C 180,E1 -2855.494,E2 -2855.494} C_VEL
LIN {X 0,Y 559.146,Z 370.835,A -85,B 0,C 180,E1 -2858.446,E2 -2858.446} C_VEL
LIN {X 0,Y 559.156,Z 370.835,A -85,B 0,C 180,E1 -2860.926,E2 -2860.926} C_VEL
LIN {X 0,Y 559.152,Z 370.834,A -85,B 0,C 180,E1 -2863.947,E2 -2863.947} C_VEL
LIN {X 0,Y 559.16,Z 370.835,A -85,B 0,C 180,E1 -2866.184,E2 -2866.184} C_VEL
LIN {X 0,Y 559.196,Z 370.829,A -85,B 0,C 180,E1 -2869.134,E2 -2869.134} C_VEL
LIN {X 0,Y 559.194,Z 370.829,A -85,B 0,C 180,E1 -2872.054,E2 -2872.054} C_VEL
LIN {X 0,Y 559.247,Z 370.823,A -85,B 0,C 180,E1 -2874.953,E2 -2874.953} C_VEL
LIN {X 0,Y 559.244,Z 370.825,A -85,B 0,C 180,E1 -2877.839,E2 -2877.839} C_VEL
LIN {X 0,Y 559.262,Z 370.825,A -85,B 0,C 180,E1 -2880.72,E2 -2880.72} C_VEL
LIN {X 0,Y 559.23,Z 370.825,A -85,B 0,C 180,E1 -2882.881,E2 -2882.881} C_VEL
LIN {X 0,Y 559.213,Z 370.828,A -85,B 0,C 180,E1 -2885.77,E2 -2885.77} C_VEL
LIN {X 0,Y 559.172,Z 370.834,A -85,B 0,C 180,E1 -2888.675,E2 -2888.675} C_VEL
LIN {X 0,Y 559.188,Z 370.834,A -85,B 0,C 180,E1 -2891.601,E2 -2891.601} C_VEL
LIN {X 0,Y 559.178,Z 370.833,A -85,B 0,C 180,E1 -2894.596,E2 -2894.596} C_VEL
LIN {X 0,Y 559.146,Z 370.835,A -85,B 0,C 180,E1 -2897.557,E2 -2897.557} C_VEL
LIN {X 0,Y 559.157,Z 370.837,A -85,B 0,C 180,E1 -2899.838,E2 -2899.838} C_VEL
LIN {X 0,Y 559.146,Z 370.838,A -85,B 0,C 180,E1 -2902.153,E2 -2902.153} C_VEL
LIN {X 0,Y 559.149,Z 370.836,A -85,B 0,C 180,E1 -2904.506,E2 -2904.506} C_VEL
LIN {X 0,Y 559.162,Z 370.834,A -85,B 0,C 180,E1 -2906.903,E2 -2906.903} C_VEL
LIN {X 0,Y 559.132,Z 370.838,A -85,B 0,C 180,E1 -2909.859,E2 -2909.859} C_VEL
LIN {X 0,Y 559.16,Z 370.834,A -85,B 0,C 180,E1 -2912.715,E2 -2912.715} C_VEL
LIN {X 0,Y 559.143,Z 370.836,A -85,B 0,C 180,E1 -2915.323,E2 -2915.323} C_VEL
LIN {X 0,Y 559.118,Z 370.839,A -85,B 0,C 180,E1 -2918.019,E2 -2918.019} C_VEL
LIN {X 0,Y 559.184,Z 370.833,A -85,B 0,C 180,E1 -2921.057,E2 -2921.057} C_VEL
LIN {X 0,Y 559.128,Z 370.841,A -85,B 0,C 180,E1 -2923.735,E2 -2923.735} C_VEL
LIN {X 0,Y 559.155,Z 370.84,A -85,B 0,C 180,E1 -2926.803,E2 -2926.803} C_VEL
LIN {X 0,Y 559.17,Z 370.836,A -85,B 0,C 180,E1 -2929.192,E2 -2929.192} C_VEL
LIN {X 0,Y 559.125,Z 370.842,A -85,B 0,C 180,E1 -2931.984,E2 -2931.984} C_VEL
LIN {X 0,Y 559.187,Z 371,A -85,B 0,C 180,E1 -2932.8,E2 -2932.8} C_VEL
LIN {X 0,Y 559.879,Z 375.253,A -85,B 0,C 180,E1 -2934.292,E2 -2934.292} C_VEL
LIN {X 0,Y 559.853,Z 381.867,A -85,B 0,C 180,E1 -2936.474,E2 -2936.474} C_VEL
LIN {X 0,Y 559.653,Z 389.811,A -85,B 0,C 180,E1 -2939.014,E2 -2939.014} C_VEL
LIN {X 0,Y 559.545,Z 399.164,A -85,B 0,C 180,E1 -2941.929,E2 -2941.929} C_VEL
LIN {X 0,Y 559.394,Z 408.52,A -85,B 0,C 180,E1 -2944.767,E2 -2944.767} C_VEL
LIN {X 0,Y 559.301,Z 417.612,A -85,B 0,C 180,E1 -2947.467,E2 -2947.467} C_VEL
LIN {X 0,Y 559.174,Z 428.042,A -85,B 0,C 180,E1 -2950.5,E2 -2950.5} C_VEL
LIN {X 0,Y 559.055,Z 438.794,A -85,B 0,C 180,E1 -2953.571,E2 -2953.571} C_VEL
LIN {X 0,Y 558.962,Z 449.385,A -85,B 0,C 180,E1 -2956.551,E2 -2956.551} C_VEL
LIN {X 0,Y 558.938,Z 451.536,A -85,B 0,C 180,E1 -2957.152,E2 -2957.152} C_VEL
LIN {X 0,Y 560.028,Z 459.592,A -85,B 0,C 180,E1 -2957.338,E2 -2957.338} C_VEL
LIN {X 0,Y 559.901,Z 471.925,A -85,B 0,C 180,E1 -2957.681,E2 -2957.681} C_VEL
LIN {X 0,Y 559.723,Z 484.318,A -85,B 0,C 180,E1 -2958.172,E2 -2958.172} C_VEL
LIN {X 0,Y 559.537,Z 496.816,A -85,B 0,C 180,E1 -2958.834,E2 -2958.834} C_VEL
LIN {X 0,Y 559.435,Z 507.949,A -85,B 0,C 180,E1 -2959.598,E2 -2959.598} C_VEL
LIN {X 0,Y 559.243,Z 517.618,A -85,B 0,C 180,E1 -2960.416,E2 -2960.416} C_VEL
LIN {X 0,Y 559.126,Z 526.427,A -85,B 0,C 180,E1 -2961.326,E2 -2961.326} C_VEL
LIN {X 0,Y 558.995,Z 535.011,A -85,B 0,C 180,E1 -2962.416,E2 -2962.416} C_VEL
LIN {X 0,Y 558.883,Z 542.695,A -85,B 0,C 180,E1 -2963.65,E2 -2963.65} C_VEL
LIN {X 0,Y 558.868,Z 547.372,A -85,B 0,C 180,E1 -2964.59,E2 -2964.59} C_VEL
LIN {X 0,Y 558.868,Z 551.682,A -85,B 0,C 180,E1 -2965.674,E2 -2965.674} C_VEL
LIN {X 0,Y 558.836,Z 553.961,A -85,B 0,C 180,E1 -2966.396,E2 -2966.396} C_VEL
LIN {X 0,Y 558.799,Z 555.812,A -85,B 0,C 180,E1 -2967.118,E2 -2967.118} C_VEL
LIN {X 0,Y 558.746,Z 557.202,A -85,B 0,C 180,E1 -2967.839,E2 -2967.839} C_VEL
LIN {X 0,Y 558.741,Z 558.785,A -85,B 0,C 180,E1 -2969.281,E2 -2969.281} C_VEL
LIN {X 0,Y 558.74,Z 559,A -85,B 0,C 180,E1 -2970.001,E2 -2970.001} C_VEL
LIN {X 0,Y 558.745,Z 558.184,A -85,B 0,C 180,E1 -2971.443,E2 -2971.443} C_VEL
LIN {X 0,Y 558.746,Z 557.198,A -85,B 0,C 180,E1 -2972.164,E2 -2972.164} C_VEL
LIN {X 0,Y 558.799,Z 555.807,A -85,B 0,C 180,E1 -2972.885,E2 -2972.885} C_VEL
LIN {X 0,Y 558.844,Z 552.892,A -85,B 0,C 180,E1 -2973.967,E2 -2973.967} C_VEL
LIN {X 0,Y 558.798,Z 548.944,A -85,B 0,C 180,E1 -2975.052,E2 -2975.052} C_VEL
LIN {X 0,Y 558.922,Z 543.86,A -85,B 0,C 180,E1 -2976.137,E2 -2976.137} C_VEL
LIN {X 0,Y 558.979,Z 537.461,A -85,B 0,C 180,E1 -2977.224,E2 -2977.224} C_VEL
LIN {X 0,Y 559.097,Z 529.468,A -85,B 0,C 180,E1 -2978.313,E2 -2978.313} C_VEL
LIN {X 0,Y 559.196,Z 521.325,A -85,B 0,C 180,E1 -2979.222,E2 -2979.222} C_VEL
LIN {X 0,Y 559.348,Z 511.388,A -85,B 0,C 180,E1 -2980.133,E2 -2980.133} C_VEL
LIN {X 0,Y 559.528,Z 500.404,A -85,B 0,C 180,E1 -2980.937,E2 -2980.937} C_VEL
LIN {X 0,Y 559.638,Z 488.801,A -85,B 0,C 180,E1 -2981.611,E2 -2981.611} C_VEL
LIN {X 0,Y 559.82,Z 476.959,A -85,B 0,C 180,E1 -2982.14,E2 -2982.14} C_VEL
LIN {X 0,Y 559.971,Z 464.132,A -85,B 0,C 180,E1 -2982.551,E2 -2982.551} C_VEL
LIN {X 0,Y 559.811,Z 457.044,A -85,B 0,C 180,E1 -2982.718,E2 -2982.718} C_VEL
LIN {X 0,Y 558.941,Z 451.526,A -85,B 0,C 180,E1 -2982.851,E2 -2982.851} C_VEL
LIN {X 0,Y 559.055,Z 441.432,A -85,B 0,C 180,E1 -2985.682,E2 -2985.682} C_VEL
LIN {X 0,Y 559.143,Z 430.841,A -85,B 0,C 180,E1 -2988.695,E2 -2988.695} C_VEL
LIN {X 0,Y 559.226,Z 420.917,A -85,B 0,C 180,E1 -2991.567,E2 -2991.567} C_VEL
LIN {X 0,Y 559.392,Z 409.747,A -85,B 0,C 180,E1 -2994.865,E2 -2994.865} C_VEL
LIN {X 0,Y 559.506,Z 400.392,A -85,B 0,C 180,E1 -2997.696,E2 -2997.696} C_VEL
LIN {X 0,Y 559.64,Z 391.124,A -85,B 0,C 180,E1 -3000.572,E2 -3000.572} C_VEL
LIN {X 0,Y 559.798,Z 383.183,A -85,B 0,C 180,E1 -3003.102,E2 -3003.102} C_VEL
LIN {X 0,Y 559.876,Z 376.383,A -85,B 0,C 180,E1 -3005.32,E2 -3005.32} C_VEL
LIN {X 0,Y 559.206,Z 370.912,A -85,B 0,C 180,E1 -3007.202,E2 -3007.202} C_VEL
LIN {X 0,Y 559.165,Z 370.836,A -85,B 0,C 180,E1 -3009.942,E2 -3009.942} C_VEL
LIN {X 0,Y 559.163,Z 370.836,A -85,B 0,C 180,E1 -3012.744,E2 -3012.744} C_VEL
LIN {X 0,Y 559.152,Z 370.837,A -85,B 0,C 180,E1 -3015.762,E2 -3015.762} C_VEL
LIN {X 0,Y 559.168,Z 370.835,A -85,B 0,C 180,E1 -3018.23,E2 -3018.23} C_VEL
LIN {X 0,Y 559.177,Z 370.833,A -85,B 0,C 180,E1 -3021.192,E2 -3021.192} C_VEL
LIN {X 0,Y 559.144,Z 370.839,A -85,B 0,C 180,E1 -3023.789,E2 -3023.789} C_VEL
LIN {X 0,Y 559.152,Z 370.836,A -85,B 0,C 180,E1 -3026.424,E2 -3026.424} C_VEL
LIN {X 0,Y 559.16,Z 370.838,A -85,B 0,C 180,E1 -3028.981,E2 -3028.981} C_VEL
LIN {X 0,Y 559.173,Z 370.833,A -85,B 0,C 180,E1 -3031.619,E2 -3031.619} C_VEL
LIN {X 0,Y 559.184,Z 370.832,A -85,B 0,C 180,E1 -3033.903,E2 -3033.903} C_VEL
LIN {X 0,Y 559.145,Z 370.838,A -85,B 0,C 180,E1 -3036.571,E2 -3036.571} C_VEL
LIN {X 0,Y 559.183,Z 370.834,A -85,B 0,C 180,E1 -3039.395,E2 -3039.395} C_VEL
LIN {X 0,Y 559.15,Z 370.837,A -85,B 0,C 180,E1 -3041.686,E2 -3041.686} C_VEL
LIN {X 0,Y 559.169,Z 370.834,A -85,B 0,C 180,E1 -3043.948,E2 -3043.948} C_VEL
LIN {X 0,Y 559.176,Z 370.834,A -85,B 0,C 180,E1 -3046.184,E2 -3046.184} C_VEL
LIN {X 0,Y 559.198,Z 370.83,A -85,B 0,C 180,E1 -3049.133,E2 -3049.133} C_VEL
LIN {X 0,Y 559.209,Z 370.83,A -85,B 0,C 180,E1 -3052.054,E2 -3052.054} C_VEL
LIN {X 0,Y 559.253,Z 370.825,A -85,B 0,C 180,E1 -3054.953,E2 -3054.953} C_VEL
LIN {X 0,Y 559.256,Z 370.824,A -85,B 0,C 180,E1 -3057.839,E2 -3057.839} C_VEL
LIN {X 0,Y 559.273,Z 370.821,A -85,B 0,C 180,E1 -3060.72,E2 -3060.72} C_VEL
LIN {X 0,Y 559.242,Z 370.825,A -85,B 0,C 180,E1 -3062.881,E2 -3062.881} C_VEL
LIN {X 0,Y 559.231,Z 370.827,A -85,B 0,C 180,E1 -3065.77,E2 -3065.77} C_VEL
LIN {X 0,Y 559.195,Z 370.831,A -85,B 0,C 180,E1 -3068.674,E2 -3068.674} C_VEL
LIN {X 0,Y 559.209,Z 370.831,A -85,B 0,C 180,E1 -3071.6,E2 -3071.6} C_VEL
LIN {X 0,Y 559.204,Z 370.831,A -85,B 0,C 180,E1 -3074.595,E2 -3074.595} C_VEL
LIN {X 0,Y 559.162,Z 370.837,A -85,B 0,C 180,E1 -3077.557,E2 -3077.557} C_VEL
LIN {X 0,Y 559.169,Z 370.836,A -85,B 0,C 180,E1 -3079.837,E2 -3079.837} C_VEL
LIN {X 0,Y 559.144,Z 370.838,A -85,B 0,C 180,E1 -3082.153,E2 -3082.153} C_VEL
LIN {X 0,Y 559.179,Z 370.834,A -85,B 0,C 180,E1 -3085.298,E2 -3085.298} C_VEL
LIN {X 0,Y 559.185,Z 370.833,A -85,B 0,C 180,E1 -3087.712,E2 -3087.712} C_VEL
LIN {X 0,Y 559.144,Z 370.837,A -85,B 0,C 180,E1 -3090.619,E2 -3090.619} C_VEL
LIN {X 0,Y 558.482,Z 370.922,A -85,B 0,C 180,E1 -3091.22,E2 -3091.22} C_VEL
LIN {X 0,Y 555.618,Z 371.278,A -85,B 0,C 180,E1 -3092.196,E2 -3092.196} C_VEL
LIN {X 0,Y 553.205,Z 371.577,A -85,B 0,C 180,E1 -3092.982,E2 -3092.982} C_VEL
LIN {X 0,Y 552.186,Z 371.705,A -85,B 0,C 180,E1 -3093.588,E2 -3093.588} C_VEL
LIN {X 0,Y 552.112,Z 371.713,A -85,B 0,C 180,E1 -3093.794,E2 -3093.794} C_VEL
LIN {X 0,Y 552.109,Z 371.714,A -85,B 0,C 180,E1 -3096.747,E2 -3096.747} C_VEL
LIN {X 0,Y 552.132,Z 371.713,A -85,B 0,C 180,E1 -3099.527,E2 -3099.527} C_VEL
LIN {X 0,Y 552.134,Z 371.711,A -85,B 0,C 180,E1 -3102.425,E2 -3102.425} C_VEL
LIN {X 0,Y 552.096,Z 371.717,A -85,B 0,C 180,E1 -3105.562,E2 -3105.562} C_VEL
LIN {X 0,Y 552.135,Z 371.71,A -85,B 0,C 180,E1 -3108.555,E2 -3108.555} C_VEL
LIN {X 0,Y 552.124,Z 371.712,A -85,B 0,C 180,E1 -3111.411,E2 -3111.411} C_VEL
LIN {X 0,Y 552.091,Z 371.717,A -85,B 0,C 180,E1 -3114.156,E2 -3114.156} C_VEL
LIN {X 0,Y 552.121,Z 371.713,A -85,B 0,C 180,E1 -3116.814,E2 -3116.814} C_VEL
LIN {X 0,Y 552.105,Z 371.714,A -85,B 0,C 180,E1 -3119.39,E2 -3119.39} C_VEL
LIN {X 0,Y 552.111,Z 371.713,A -85,B 0,C 180,E1 -3121.901,E2 -3121.901} C_VEL
LIN {X 0,Y 552.161,Z 371.708,A -85,B 0,C 180,E1 -3124.649,E2 -3124.649} C_VEL
LIN {X 0,Y 552.098,Z 371.716,A -85,B 0,C 180,E1 -3127.548,E2 -3127.548} C_VEL
LIN {X 0,Y 552.151,Z 371.709,A -85,B 0,C 180,E1 -3130.374,E2 -3130.374} C_VEL
LIN {X 0,Y 552.139,Z 371.71,A -85,B 0,C 180,E1 -3132.976,E2 -3132.976} C_VEL
LIN {X 0,Y 552.142,Z 371.71,A -85,B 0,C 180,E1 -3136.003,E2 -3136.003} C_VEL
LIN {X 0,Y 552.052,Z 371.723,A -85,B 0,C 180,E1 -3138.598,E2 -3138.598} C_VEL
LIN {X 0,Y 551.919,Z 372.042,A -85,B 0,C 180,E1 -3139.73,E2 -3139.73} C_VEL
LIN {X 0,Y 551.907,Z 374.564,A -85,B 0,C 180,E1 -3141.947,E2 -3141.947} C_VEL
LIN {X 0,Y 551.914,Z 377.903,A -85,B 0,C 180,E1 -3144.885,E2 -3144.885} C_VEL
LIN {X 0,Y 551.786,Z 381.17,A -85,B 0,C 180,E1 -3147.809,E2 -3147.809} C_VEL
LIN {X 0,Y 551.804,Z 383.617,A -85,B 0,C 180,E1 -3149.999,E2 -3149.999} C_VEL
LIN {X 0,Y 551.689,Z 386.945,A -85,B 0,C 180,E1 -3152.919,E2 -3152.919} C_VEL
LIN {X 0,Y 551.658,Z 389.391,A -85,B 0,C 180,E1 -3155.115,E2 -3155.115} C_VEL
LIN {X 0,Y 551.684,Z 392.129,A -85,B 0,C 180,E1 -3157.317,E2 -3157.317} C_VEL
LIN {X 0,Y 551.673,Z 395.769,A -85,B 0,C 180,E1 -3160.11,E2 -3160.11} C_VEL
LIN {X 0,Y 553.01,Z 404.356,A -85,B 0,C 180,E1 -3160.34,E2 -3160.34} C_VEL
LIN {X 0,Y 552.912,Z 417.117,A -85,B 0,C 180,E1 -3160.758,E2 -3160.758} C_VEL
LIN {X 0,Y 552.678,Z 428.872,A -85,B 0,C 180,E1 -3161.29,E2 -3161.29} C_VEL
LIN {X 0,Y 552.521,Z 439.783,A -85,B 0,C 180,E1 -3161.927,E2 -3161.927} C_VEL
LIN {X 0,Y 552.324,Z 450.099,A -85,B 0,C 180,E1 -3162.678,E2 -3162.678} C_VEL
LIN {X 0,Y 552.185,Z 458.583,A -85,B 0,C 180,E1 -3163.43,E2 -3163.43} C_VEL
LIN {X 0,Y 552.032,Z 466.863,A -85,B 0,C 180,E1 -3164.308,E2 -3164.308} C_VEL
LIN {X 0,Y 551.938,Z 474.711,A -85,B 0,C 180,E1 -3165.319,E2 -3165.319} C_VEL
LIN {X 0,Y 551.833,Z 481.85,A -85,B 0,C 180,E1 -3166.46,E2 -3166.46} C_VEL
LIN {X 0,Y 551.788,Z 486.911,A -85,B 0,C 180,E1 -3167.46,E2 -3167.46} C_VEL
LIN {X 0,Y 551.726,Z 491.358,A -85,B 0,C 180,E1 -3168.568,E2 -3168.568} C_VEL
LIN {X 0,Y 551.694,Z 494.249,A -85,B 0,C 180,E1 -3169.493,E2 -3169.493} C_VEL
LIN {X 0,Y 551.661,Z 495.795,A -85,B 0,C 180,E1 -3170.117,E2 -3170.117} C_VEL
LIN {X 0,Y 551.667,Z 498.165,A -85,B 0,C 180,E1 -3171.567,E2 -3171.567} C_VEL
LIN {X 0,Y 551.641,Z 498.876,A -85,B 0,C 180,E1 -3172.468,E2 -3172.468} C_VEL
LIN {X 0,Y 551.655,Z 498.914,A -85,B 0,C 180,E1 -3173.47,E2 -3173.47} C_VEL
LIN {X 0,Y 551.652,Z 497.77,A -85,B 0,C 180,E1 -3174.859,E2 -3174.859} C_VEL
LIN {X 0,Y 551.645,Z 496.41,A -85,B 0,C 180,E1 -3175.666,E2 -3175.666} C_VEL
LIN {X 0,Y 551.72,Z 493.326,A -85,B 0,C 180,E1 -3176.914,E2 -3176.914} C_VEL
LIN {X 0,Y 551.762,Z 489.124,A -85,B 0,C 180,E1 -3178.115,E2 -3178.115} C_VEL
LIN {X 0,Y 551.84,Z 483.336,A -85,B 0,C 180,E1 -3179.359,E2 -3179.359} C_VEL
LIN {X 0,Y 551.958,Z 475.757,A -85,B 0,C 180,E1 -3180.616,E2 -3180.616} C_VEL
LIN {X 0,Y 552.033,Z 467.762,A -85,B 0,C 180,E1 -3181.677,E2 -3181.677} C_VEL
LIN {X 0,Y 552.241,Z 458.36,A -85,B 0,C 180,E1 -3182.681,E2 -3182.681} C_VEL
LIN {X 0,Y 552.397,Z 447.697,A -85,B 0,C 180,E1 -3183.601,E2 -3183.601} C_VEL
LIN {X 0,Y 552.564,Z 437.468,A -85,B 0,C 180,E1 -3184.313,E2 -3184.313} C_VEL
LIN {X 0,Y 552.757,Z 425.863,A -85,B 0,C 180,E1 -3184.951,E2 -3184.951} C_VEL
LIN {X 0,Y 552.894,Z 413.66,A -85,B 0,C 180,E1 -3185.461,E2 -3185.461} C_VEL
LIN {X 0,Y 552.903,Z 402.813,A -85,B 0,C 180,E1 -3185.793,E2 -3185.793} C_VEL
LIN {X 0,Y 551.674,Z 395.675,A -85,B 0,C 180,E1 -3185.993,E2 -3185.993} C_VEL
LIN {X 0,Y 551.65,Z 391.842,A -85,B 0,C 180,E1 -3189.001,E2 -3189.001} C_VEL
LIN {X 0,Y 551.692,Z 388.849,A -85,B 0,C 180,E1 -3191.482,E2 -3191.482} C_VEL
LIN {X 0,Y 551.757,Z 385.535,A -85,B 0,C 180,E1 -3194.496,E2 -3194.496} C_VEL
LIN {X 0,Y 551.765,Z 383.214,A -85,B 0,C 180,E1 -3196.551,E2 -3196.551} C_VEL
LIN {X 0,Y 551.795,Z 379.996,A -85,B 0,C 180,E1 -3199.491,E2 -3199.491} C_VEL
LIN {X 0,Y 551.85,Z 376.851,A -85,B 0,C 180,E1 -3202.317,E2 -3202.317} C_VEL
LIN {X 0,Y 551.87,Z 373.784,A -85,B 0,C 180,E1 -3205.035,E2 -3205.035} C_VEL
LIN {X 0,Y 551.909,Z 371.784,A -85,B 0,C 180,E1 -3206.8,E2 -3206.8} C_VEL
LIN {X 0,Y 552.09,Z 371.717,A -85,B 0,C 180,E1 -3209.39,E2 -3209.39} C_VEL
LIN {X 0,Y 552.11,Z 371.712,A -85,B 0,C 180,E1 -3211.902,E2 -3211.902} C_VEL
LIN {X 0,Y 552.137,Z 371.709,A -85,B 0,C 180,E1 -3214.648,E2 -3214.648} C_VEL
LIN {X 0,Y 552.106,Z 371.715,A -85,B 0,C 180,E1 -3217.55,E2 -3217.55} C_VEL
LIN {X 0,Y 552.139,Z 371.71,A -85,B 0,C 180,E1 -3220.674,E2 -3220.674} C_VEL
LIN {X 0,Y 552.101,Z 371.713,A -85,B 0,C 180,E1 -3223.737,E2 -3223.737} C_VEL
LIN {X 0,Y 552.121,Z 371.713,A -85,B 0,C 180,E1 -3226.004,E2 -3226.004} C_VEL
LIN {X 0,Y 552.162,Z 371.706,A -85,B 0,C 180,E1 -3228.993,E2 -3228.993} C_VEL
LIN {X 0,Y 552.147,Z 371.707,A -85,B 0,C 180,E1 -3231.951,E2 -3231.951} C_VEL
LIN {X 0,Y 552.222,Z 371.698,A -85,B 0,C 180,E1 -3234.889,E2 -3234.889} C_VEL
LIN {X 0,Y 552.214,Z 371.7,A -85,B 0,C 180,E1 -3237.812,E2 -3237.812} C_VEL
LIN {X 0,Y 552.231,Z 371.701,A -85,B 0,C 180,E1 -3240.729,E2 -3240.729} C_VEL
LIN {X 0,Y 552.196,Z 371.701,A -85,B 0,C 180,E1 -3242.918,E2 -3242.918} C_VEL
LIN {X 0,Y 552.183,Z 371.704,A -85,B 0,C 180,E1 -3245.844,E2 -3245.844} C_VEL
LIN {X 0,Y 552.143,Z 371.711,A -85,B 0,C 180,E1 -3248.786,E2 -3248.786} C_VEL
LIN {X 0,Y 552.144,Z 371.71,A -85,B 0,C 180,E1 -3251.751,E2 -3251.751} C_VEL
LIN {X 0,Y 552.116,Z 371.711,A -85,B 0,C 180,E1 -3254.749,E2 -3254.749} C_VEL
LIN {X 0,Y 552.098,Z 371.713,A -85,B 0,C 180,E1 -3257.789,E2 -3257.789} C_VEL
LIN {X 0,Y 552.116,Z 371.712,A -85,B 0,C 180,E1 -3260.102,E2 -3260.102} C_VEL
LIN {X 0,Y 552.107,Z 371.717,A -85,B 0,C 180,E1 -3262.45,E2 -3262.45} C_VEL
LIN {X 0,Y 552.138,Z 371.711,A -85,B 0,C 180,E1 -3265.352,E2 -3265.352} C_VEL
LIN {X 0,Y 552.11,Z 371.714,A -85,B 0,C 180,E1 -3268.098,E2 -3268.098} C_VEL
LIN {X 0,Y 552.091,Z 371.718,A -85,B 0,C 180,E1 -3270.61,E2 -3270.61} C_VEL
LIN {X 0,Y 552.107,Z 371.717,A -85,B 0,C 180,E1 -3273.187,E2 -3273.187} C_VEL
LIN {X 0,Y 552.098,Z 371.717,A -85,B 0,C 180,E1 -3275.843,E2 -3275.843} C_VEL
LIN {X 0,Y 552.108,Z 371.713,A -85,B 0,C 180,E1 -3279.063,E2 -3279.063} C_VEL
LIN {X 0,Y 552.157,Z 371.711,A -85,B 0,C 180,E1 -3281.443,E2 -3281.443} C_VEL
LIN {X 0,Y 552.082,Z 371.718,A -85,B 0,C 180,E1 -3284.534,E2 -3284.534} C_VEL
LIN {X 0,Y 552.12,Z 371.713,A -85,B 0,C 180,E1 -3287.586,E2 -3287.586} C_VEL
LIN {X 0,Y 552.125,Z 371.713,A -85,B 0,C 180,E1 -3290.475,E2 -3290.475} C_VEL
LIN {X 0,Y 552.119,Z 371.774,A -85,B 0,C 180,E1 -3292.514,E2 -3292.514} C_VEL
LIN {X 0,Y 552.94,Z 376.58,A -85,B 0,C 180,E1 -3294.223,E2 -3294.223} C_VEL
LIN {X 0,Y 552.846,Z 384.515,A -85,B 0,C 180,E1 -3296.866,E2 -3296.866} C_VEL
LIN {X 0,Y 552.66,Z 392.458,A -85,B 0,C 180,E1 -3299.427,E2 -3299.427} C_VEL
LIN {X 0,Y 552.512,Z 401.726,A -85,B 0,C 180,E1 -3302.338,E2 -3302.338} C_VEL
LIN {X 0,Y 552.36,Z 410.993,A -85,B 0,C 180,E1 -3305.175,E2 -3305.175} C_VEL
LIN {X 0,Y 552.249,Z 420.261,A -85,B 0,C 180,E1 -3307.952,E2 -3307.952} C_VEL
LIN {X 0,Y 552.086,Z 430.851,A -85,B 0,C 180,E1 -3311.06,E2 -3311.06} C_VEL
LIN {X 0,Y 551.993,Z 441.442,A -85,B 0,C 180,E1 -3314.115,E2 -3314.115} C_VEL
LIN {X 0,Y 551.888,Z 451.536,A -85,B 0,C 180,E1 -3316.985,E2 -3316.985} C_VEL
LIN {X 0,Y 553.098,Z 460.589,A -85,B 0,C 180,E1 -3317.2,E2 -3317.2} C_VEL
LIN {X 0,Y 552.94,Z 473.225,A -85,B 0,C 180,E1 -3317.57,E2 -3317.57} C_VEL
LIN {X 0,Y 552.749,Z 485.521,A -85,B 0,C 180,E1 -3318.078,E2 -3318.078} C_VEL
LIN {X 0,Y 552.567,Z 497.222,A -85,B 0,C 180,E1 -3318.717,E2 -3318.717} C_VEL
LIN {X 0,Y 552.431,Z 507.948,A -85,B 0,C 180,E1 -3319.464,E2 -3319.464} C_VEL
LIN {X 0,Y 552.232,Z 517.618,A -85,B 0,C 180,E1 -3320.294,E2 -3320.294} C_VEL
LIN {X 0,Y 552.078,Z 526.427,A -85,B 0,C 180,E1 -3321.215,E2 -3321.215} C_VEL
LIN {X 0,Y 551.948,Z 535.011,A -85,B 0,C 180,E1 -3322.318,E2 -3322.318} C_VEL
LIN {X 0,Y 551.821,Z 541.876,A -85,B 0,C 180,E1 -3323.42,E2 -3323.42} C_VEL
LIN {X 0,Y 551.803,Z 547.372,A -85,B 0,C 180,E1 -3324.52,E2 -3324.52} C_VEL
LIN {X 0,Y 551.764,Z 551.683,A -85,B 0,C 180,E1 -3325.618,E2 -3325.618} C_VEL
LIN {X 0,Y 551.75,Z 553.961,A -85,B 0,C 180,E1 -3326.35,E2 -3326.35} C_VEL
LIN {X 0,Y 551.723,Z 555.812,A -85,B 0,C 180,E1 -3327.081,E2 -3327.081} C_VEL
LIN {X 0,Y 551.645,Z 558.187,A -85,B 0,C 180,E1 -3328.541,E2 -3328.541} C_VEL
LIN {X 0,Y 551.64,Z 559,A -85,B 0,C 180,E1 -3330.001,E2 -3330.001} C_VEL
LIN {X 0,Y 551.645,Z 558.184,A -85,B 0,C 180,E1 -3331.461,E2 -3331.461} C_VEL
LIN {X 0,Y 551.657,Z 557.198,A -85,B 0,C 180,E1 -3332.192,E2 -3332.192} C_VEL
LIN {X 0,Y 551.724,Z 555.807,A -85,B 0,C 180,E1 -3332.922,E2 -3332.922} C_VEL
LIN {X 0,Y 551.764,Z 552.892,A -85,B 0,C 180,E1 -3334.018,E2 -3334.018} C_VEL
LIN {X 0,Y 551.724,Z 548.944,A -85,B 0,C 180,E1 -3335.117,E2 -3335.117} C_VEL
LIN {X 0,Y 551.825,Z 543.189,A -85,B 0,C 180,E1 -3336.341,E2 -3336.341} C_VEL
LIN {X 0,Y 551.928,Z 536.229,A -85,B 0,C 180,E1 -3337.501,E2 -3337.501} C_VEL
LIN {X 0,Y 552.079,Z 527.98,A -85,B 0,C 180,E1 -3338.604,E2 -3338.604} C_VEL
LIN {X 0,Y 552.202,Z 519.525,A -85,B 0,C 180,E1 -3339.525,E2 -3339.525} C_VEL
LIN {X 0,Y 552.406,Z 509.081,A -85,B 0,C 180,E1 -3340.446,E2 -3340.446} C_VEL
LIN {X 0,Y 552.578,Z 498.348,A -85,B 0,C 180,E1 -3341.21,E2 -3341.21} C_VEL
LIN {X 0,Y 552.702,Z 487.389,A -85,B 0,C 180,E1 -3341.833,E2 -3341.833} C_VEL
LIN {X 0,Y 552.913,Z 475.731,A -85,B 0,C 180,E1 -3342.341,E2 -3342.341} C_VEL
LIN {X 0,Y 553.07,Z 462.304,A -85,B 0,C 180,E1 -3342.757,E2 -3342.757} C_VEL
LIN {X 0,Y 552.765,Z 457.044,A -85,B 0,C 180,E1 -3342.883,E2 -3342.883} C_VEL
LIN {X 0,Y 551.89,Z 451.526,A -85,B 0,C 180,E1 -3343.018,E2 -3343.018} C_VEL
LIN {X 0,Y 551.996,Z 441.432,A -85,B 0,C 180,E1 -3345.888,E2 -3345.888} C_VEL
LIN {X 0,Y 552.093,Z 430.841,A -85,B 0,C 180,E1 -3348.943,E2 -3348.943} C_VEL
LIN {X 0,Y 552.255,Z 420.251,A -85,B 0,C 180,E1 -3352.051,E2 -3352.051} C_VEL
LIN {X 0,Y 552.365,Z 410.983,A -85,B 0,C 180,E1 -3354.828,E2 -3354.828} C_VEL
LIN {X 0,Y 552.509,Z 401.715,A -85,B 0,C 180,E1 -3357.665,E2 -3357.665} C_VEL
LIN {X 0,Y 552.67,Z 392.448,A -85,B 0,C 180,E1 -3360.575,E2 -3360.575} C_VEL
LIN {X 0,Y 552.855,Z 384.505,A -85,B 0,C 180,E1 -3363.137,E2 -3363.137} C_VEL
LIN {X 0,Y 552.922,Z 377.111,A -85,B 0,C 180,E1 -3365.562,E2 -3365.562} C_VEL
LIN {X 0,Y 552.134,Z 371.713,A -85,B 0,C 180,E1 -3367.489,E2 -3367.489} C_VEL
LIN {X 0,Y 552.114,Z 371.715,A -85,B 0,C 180,E1 -3370.482,E2 -3370.482} C_VEL
LIN {X 0,Y 552.112,Z 371.716,A -85,B 0,C 180,E1 -3373.424,E2 -3373.424} C_VEL
LIN {X 0,Y 552.112,Z 371.716,A -85,B 0,C 180,E1 -3376.577,E2 -3376.577} C_VEL
LIN {X 0,Y 552.113,Z 371.715,A -85,B 0,C 180,E1 -3379.519,E2 -3379.519} C_VEL
LIN {X 0,Y 552.096,Z 371.715,A -85,B 0,C 180,E1 -3382.336,E2 -3382.336} C_VEL
LIN {X 0,Y 552.087,Z 371.717,A -85,B 0,C 180,E1 -3385.051,E2 -3385.051} C_VEL
LIN {X 0,Y 552.119,Z 371.713,A -85,B 0,C 180,E1 -3387.681,E2 -3387.681} C_VEL
LIN {X 0,Y 552.116,Z 371.714,A -85,B 0,C 180,E1 -3390.235,E2 -3390.235} C_VEL
LIN {X 0,Y 552.142,Z 371.711,A -85,B 0,C 180,E1 -3393,E2 -3393} C_VEL
LIN {X 0,Y 552.117,Z 371.715,A -85,B 0,C 180,E1 -3395.161,E2 -3395.161} C_VEL
LIN {X 0,Y 552.13,Z 371.714,A -85,B 0,C 180,E1 -3398.337,E2 -3398.337} C_VEL
LIN {X 0,Y 552.16,Z 371.708,A -85,B 0,C 180,E1 -3400.674,E2 -3400.674} C_VEL
LIN {X 0,Y 552.12,Z 371.713,A -85,B 0,C 180,E1 -3403.737,E2 -3403.737} C_VEL
LIN {X 0,Y 552.14,Z 371.71,A -85,B 0,C 180,E1 -3406.004,E2 -3406.004} C_VEL
LIN {X 0,Y 552.166,Z 371.706,A -85,B 0,C 180,E1 -3408.993,E2 -3408.993} C_VEL
LIN {X 0,Y 552.163,Z 371.709,A -85,B 0,C 180,E1 -3411.952,E2 -3411.952} C_VEL
LIN {X 0,Y 552.229,Z 371.7,A -85,B 0,C 180,E1 -3414.889,E2 -3414.889} C_VEL
LIN {X 0,Y 552.227,Z 371.7,A -85,B 0,C 180,E1 -3417.812,E2 -3417.812} C_VEL
LIN {X 0,Y 552.243,Z 371.697,A -85,B 0,C 180,E1 -3420.729,E2 -3420.729} C_VEL
LIN {X 0,Y 552.208,Z 371.702,A -85,B 0,C 180,E1 -3422.918,E2 -3422.918} C_VEL
LIN {X 0,Y 552.201,Z 371.702,A -85,B 0,C 180,E1 -3425.844,E2 -3425.844} C_VEL
LIN {X 0,Y 552.165,Z 371.706,A -85,B 0,C 180,E1 -3428.786,E2 -3428.786} C_VEL
LIN {X 0,Y 552.167,Z 371.707,A -85,B 0,C 180,E1 -3431.75,E2 -3431.75} C_VEL
LIN {X 0,Y 552.14,Z 371.711,A -85,B 0,C 180,E1 -3434.748,E2 -3434.748} C_VEL
LIN {X 0,Y 552.112,Z 371.715,A -85,B 0,C 180,E1 -3437.788,E2 -3437.788} C_VEL
LIN {X 0,Y 552.13,Z 371.711,A -85,B 0,C 180,E1 -3440.101,E2 -3440.101} C_VEL
LIN {X 0,Y 552.096,Z 371.715,A -85,B 0,C 180,E1 -3442.451,E2 -3442.451} C_VEL
LIN {X 0,Y 552.159,Z 371.708,A -85,B 0,C 180,E1 -3445.35,E2 -3445.35} C_VEL
LIN {X 0,Y 552.124,Z 371.713,A -85,B 0,C 180,E1 -3448.098,E2 -3448.098} C_VEL
LIN {X 0,Y 552.107,Z 371.713,A -85,B 0,C 180,E1 -3450.615,E2 -3450.615} C_VEL
LIN {X 0,Y 552.116,Z 371.715,A -85,B 0,C 180,E1 -3453.186,E2 -3453.186} C_VEL
LIN {X 0,Y 552.112,Z 371.713,A -85,B 0,C 180,E1 -3453.794,E2 -3453.794} C_VEL
LIN {X 0,Y 551.479,Z 371.794,A -85,B 0,C 180,E1 -3454.402,E2 -3454.402} C_VEL
LIN {X 0,Y 548.657,Z 372.146,A -85,B 0,C 180,E1 -3455.39,E2 -3455.39} C_VEL
LIN {X 0,Y 546.236,Z 372.447,A -85,B 0,C 180,E1 -3456.185,E2 -3456.185} C_VEL
LIN {X 0,Y 545.166,Z 372.579,A -85,B 0,C 180,E1 -3456.799,E2 -3456.799} C_VEL
LIN {X 0,Y 545.065,Z 372.591,A -85,B 0,C 180,E1 -3457.007,E2 -3457.007} C_VEL
LIN {X 0,Y 545.069,Z 372.591,A -85,B 0,C 180,E1 -3460.142,E2 -3460.142} C_VEL
LIN {X 0,Y 545.083,Z 372.589,A -85,B 0,C 180,E1 -3463.106,E2 -3463.106} C_VEL
LIN {X 0,Y 545.053,Z 372.591,A -85,B 0,C 180,E1 -3466.226,E2 -3466.226} C_VEL
LIN {X 0,Y 545.092,Z 372.59,A -85,B 0,C 180,E1 -3468.885,E2 -3468.885} C_VEL
LIN {X 0,Y 545.088,Z 372.59,A -85,B 0,C 180,E1 -3470.818,E2 -3470.818} C_VEL
LIN {X 0,Y 545.047,Z 372.594,A -85,B 0,C 180,E1 -3473.619,E2 -3473.619} C_VEL
LIN {X 0,Y 545.071,Z 372.591,A -85,B 0,C 180,E1 -3476.328,E2 -3476.328} C_VEL
LIN {X 0,Y 545.07,Z 372.592,A -85,B 0,C 180,E1 -3478.951,E2 -3478.951} C_VEL
LIN {X 0,Y 545.106,Z 372.586,A -85,B 0,C 180,E1 -3481.507,E2 -3481.507} C_VEL
LIN {X 0,Y 545.101,Z 372.588,A -85,B 0,C 180,E1 -3484.49,E2 -3484.49} C_VEL
LIN {X 0,Y 545.044,Z 372.595,A -85,B 0,C 180,E1 -3487.241,E2 -3487.241} C_VEL
LIN {X 0,Y 545.123,Z 372.585,A -85,B 0,C 180,E1 -3490.414,E2 -3490.414} C_VEL
LIN {X 0,Y 545.07,Z 372.592,A -85,B 0,C 180,E1 -3493.52,E2 -3493.52} C_VEL
LIN {X 0,Y 545.101,Z 372.588,A -85,B 0,C 180,E1 -3495.819,E2 -3495.819} C_VEL
LIN {X 0,Y 545.012,Z 372.6,A -85,B 0,C 180,E1 -3498.531,E2 -3498.531} C_VEL
LIN {X 0,Y 544.867,Z 372.618,A -85,B 0,C 180,E1 -3499.595,E2 -3499.595} C_VEL
LIN {X 0,Y 544.808,Z 375.927,A -85,B 0,C 180,E1 -3502.587,E2 -3502.587} C_VEL
LIN {X 0,Y 544.787,Z 379.278,A -85,B 0,C 180,E1 -3505.559,E2 -3505.559} C_VEL
LIN {X 0,Y 544.675,Z 382.6,A -85,B 0,C 180,E1 -3508.52,E2 -3508.52} C_VEL
LIN {X 0,Y 544.633,Z 385.077,A -85,B 0,C 180,E1 -3510.738,E2 -3510.738} C_VEL
LIN {X 0,Y 544.697,Z 388.397,A -85,B 0,C 180,E1 -3513.697,E2 -3513.697} C_VEL
LIN {X 0,Y 544.634,Z 391.713,A -85,B 0,C 180,E1 -3516.668,E2 -3516.668} C_VEL
LIN {X 0,Y 544.554,Z 394.391,A -85,B 0,C 180,E1 -3518.908,E2 -3518.908} C_VEL
LIN {X 0,Y 544.568,Z 395.765,A -85,B 0,C 180,E1 -3519.938,E2 -3519.938} C_VEL
LIN {X 0,Y 546.088,Z 405.792,A -85,B 0,C 180,E1 -3520.214,E2 -3520.214} C_VEL
LIN {X 0,Y 545.972,Z 418.61,A -85,B 0,C 180,E1 -3520.662,E2 -3520.662} C_VEL
LIN {X 0,Y 545.708,Z 430.061,A -85,B 0,C 180,E1 -3521.201,E2 -3521.201} C_VEL
LIN {X 0,Y 545.496,Z 441.477,A -85,B 0,C 180,E1 -3521.894,E2 -3521.894} C_VEL
LIN {X 0,Y 545.272,Z 452.544,A -85,B 0,C 180,E1 -3522.75,E2 -3522.75} C_VEL
LIN {X 0,Y 545.096,Z 461.564,A -85,B 0,C 180,E1 -3523.608,E2 -3523.608} C_VEL
LIN {X 0,Y 544.928,Z 470.91,A -85,B 0,C 180,E1 -3524.696,E2 -3524.696} C_VEL
LIN {X 0,Y 544.816,Z 479.151,A -85,B 0,C 180,E1 -3525.908,E2 -3525.908} C_VEL
LIN {X 0,Y 544.738,Z 484.475,A -85,B 0,C 180,E1 -3526.873,E2 -3526.873} C_VEL
LIN {X 0,Y 544.667,Z 489.62,A -85,B 0,C 180,E1 -3528.038,E2 -3528.038} C_VEL
LIN {X 0,Y 544.615,Z 493.571,A -85,B 0,C 180,E1 -3529.21,E2 -3529.21} C_VEL
LIN {X 0,Y 544.562,Z 496.414,A -85,B 0,C 180,E1 -3530.391,E2 -3530.391} C_VEL
LIN {X 0,Y 544.565,Z 498.316,A -85,B 0,C 180,E1 -3531.688,E2 -3531.688} C_VEL
LIN {X 0,Y 544.539,Z 498.949,A -85,B 0,C 180,E1 -3532.778,E2 -3532.778} C_VEL
LIN {X 0,Y 544.574,Z 498.883,A -85,B 0,C 180,E1 -3533.61,E2 -3533.61} C_VEL
LIN {X 0,Y 544.567,Z 498.328,A -85,B 0,C 180,E1 -3534.39,E2 -3534.39} C_VEL
LIN {X 0,Y 544.562,Z 497.001,A -85,B 0,C 180,E1 -3535.39,E2 -3535.39} C_VEL
LIN {X 0,Y 544.595,Z 494.776,A -85,B 0,C 180,E1 -3536.435,E2 -3536.435} C_VEL
LIN {X 0,Y 544.645,Z 491.033,A -85,B 0,C 180,E1 -3537.678,E2 -3537.678} C_VEL
LIN {X 0,Y 544.721,Z 485.612,A -85,B 0,C 180,E1 -3538.983,E2 -3538.983} C_VEL
LIN {X 0,Y 544.8,Z 479.024,A -85,B 0,C 180,E1 -3540.203,E2 -3540.203} C_VEL
LIN {X 0,Y 544.93,Z 471.951,A -85,B 0,C 180,E1 -3541.254,E2 -3541.254} C_VEL
LIN {X 0,Y 545.092,Z 462.86,A -85,B 0,C 180,E1 -3542.346,E2 -3542.346} C_VEL
LIN {X 0,Y 545.316,Z 452.617,A -85,B 0,C 180,E1 -3543.333,E2 -3543.333} C_VEL
LIN {X 0,Y 545.501,Z 441.483,A -85,B 0,C 180,E1 -3544.195,E2 -3544.195} C_VEL
LIN {X 0,Y 545.73,Z 429.727,A -85,B 0,C 180,E1 -3544.906,E2 -3544.906} C_VEL
LIN {X 0,Y 545.951,Z 417.759,A -85,B 0,C 180,E1 -3545.465,E2 -3545.465} C_VEL
LIN {X 0,Y 546.105,Z 405.281,A -85,B 0,C 180,E1 -3545.89,E2 -3545.89} C_VEL
LIN {X 0,Y 544.555,Z 395.662,A -85,B 0,C 180,E1 -3546.176,E2 -3546.176} C_VEL
LIN {X 0,Y 544.556,Z 391.947,A -85,B 0,C 180,E1 -3549.253,E2 -3549.253} C_VEL
LIN {X 0,Y 544.623,Z 388.797,A -85,B 0,C 180,E1 -3552.143,E2 -3552.143} C_VEL
LIN {X 0,Y 544.704,Z 385.379,A -85,B 0,C 180,E1 -3555.202,E2 -3555.202} C_VEL
LIN {X 0,Y 544.73,Z 382.448,A -85,B 0,C 180,E1 -3557.864,E2 -3557.864} C_VEL
LIN {X 0,Y 544.739,Z 379.225,A -85,B 0,C 180,E1 -3560.789,E2 -3560.789} C_VEL
LIN {X 0,Y 544.794,Z 376.078,A -85,B 0,C 180,E1 -3563.6,E2 -3563.6} C_VEL
LIN {X 0,Y 544.836,Z 373.039,A -85,B 0,C 180,E1 -3566.312,E2 -3566.312} C_VEL
LIN {X 0,Y 544.916,Z 372.613,A -85,B 0,C 180,E1 -3567.201,E2 -3567.201} C_VEL
LIN {X 0,Y 545.084,Z 372.59,A -85,B 0,C 180,E1 -3569.812,E2 -3569.812} C_VEL
LIN {X 0,Y 545.084,Z 372.588,A -85,B 0,C 180,E1 -3572.823,E2 -3572.823} C_VEL
LIN {X 0,Y 545.045,Z 372.592,A -85,B 0,C 180,E1 -3575.631,E2 -3575.631} C_VEL
LIN {X 0,Y 545.08,Z 372.589,A -85,B 0,C 180,E1 -3578.17,E2 -3578.17} C_VEL
LIN {X 0,Y 545.069,Z 372.589,A -85,B 0,C 180,E1 -3581.195,E2 -3581.195} C_VEL
LIN {X 0,Y 545.057,Z 372.591,A -85,B 0,C 180,E1 -3583.521,E2 -3583.521} C_VEL
LIN {X 0,Y 545.078,Z 372.591,A -85,B 0,C 180,E1 -3585.82,E2 -3585.82} C_VEL
LIN {X 0,Y 545.115,Z 372.585,A -85,B 0,C 180,E1 -3588.849,E2 -3588.849} C_VEL
LIN {X 0,Y 545.116,Z 372.583,A -85,B 0,C 180,E1 -3591.847,E2 -3591.847} C_VEL
LIN {X 0,Y 545.197,Z 372.573,A -85,B 0,C 180,E1 -3594.823,E2 -3594.823} C_VEL
LIN {X 0,Y 545.185,Z 372.576,A -85,B 0,C 180,E1 -3597.784,E2 -3597.784} C_VEL
LIN {X 0,Y 545.2,Z 372.576,A -85,B 0,C 180,E1 -3600.739,E2 -3600.739} C_VEL
LIN {X 0,Y 545.162,Z 372.577,A -85,B 0,C 180,E1 -3602.956,E2 -3602.956} C_VEL
LIN {X 0,Y 545.155,Z 372.58,A -85,B 0,C 180,E1 -3605.92,E2 -3605.92} C_VEL
LIN {X 0,Y 545.102,Z 372.589,A -85,B 0,C 180,E1 -3608.9,E2 -3608.9} C_VEL
LIN {X 0,Y 545.115,Z 372.584,A -85,B 0,C 180,E1 -3611.905,E2 -3611.905} C_VEL
LIN {X 0,Y 545.066,Z 372.589,A -85,B 0,C 180,E1 -3614.944,E2 -3614.944} C_VEL
LIN {X 0,Y 545.067,Z 372.591,A -85,B 0,C 180,E1 -3618.026,E2 -3618.026} C_VEL
LIN {X 0,Y 545.081,Z 372.587,A -85,B 0,C 180,E1 -3620.373,E2 -3620.373} C_VEL
LIN {X 0,Y 545.124,Z 372.585,A -85,B 0,C 180,E1 -3623.557,E2 -3623.557} C_VEL
LIN {X 0,Y 545.071,Z 372.59,A -85,B 0,C 180,E1 -3626.001,E2 -3626.001} C_VEL
LIN {X 0,Y 545.074,Z 372.59,A -85,B 0,C 180,E1 -3628.75,E2 -3628.75} C_VEL
LIN {X 0,Y 545.062,Z 372.593,A -85,B 0,C 180,E1 -3631.684,E2 -3631.684} C_VEL
LIN {X 0,Y 545.066,Z 372.594,A -85,B 0,C 180,E1 -3634.564,E2 -3634.564} C_VEL
LIN {X 0,Y 545.054,Z 372.595,A -85,B 0,C 180,E1 -3637.303,E2 -3637.303} C_VEL
LIN {X 0,Y 545.098,Z 372.587,A -85,B 0,C 180,E1 -3640.478,E2 -3640.478} C_VEL
LIN {X 0,Y 545.065,Z 372.593,A -85,B 0,C 180,E1 -3643.108,E2 -3643.108} C_VEL
LIN {X 0,Y 545.052,Z 372.594,A -85,B 0,C 180,E1 -3646.226,E2 -3646.226} C_VEL
LIN {X 0,Y 545.094,Z 372.588,A -85,B 0,C 180,E1 -3648.889,E2 -3648.889} C_VEL
LIN {X 0,Y 545.044,Z 372.596,A -85,B 0,C 180,E1 -3651.765,E2 -3651.765} C_VEL
LIN {X 0,Y 545.055,Z 372.7,A -85,B 0,C 180,E1 -3652.293,E2 -3652.293} C_VEL
LIN {X 0,Y 546.002,Z 378.006,A -85,B 0,C 180,E1 -3654.186,E2 -3654.186} C_VEL
LIN {X 0,Y 545.881,Z 385.781,A -85,B 0,C 180,E1 -3656.809,E2 -3656.809} C_VEL
LIN {X 0,Y 545.694,Z 393.599,A -85,B 0,C 180,E1 -3659.364,E2 -3659.364} C_VEL
LIN {X 0,Y 545.505,Z 403.049,A -85,B 0,C 180,E1 -3662.369,E2 -3662.369} C_VEL
LIN {X 0,Y 545.35,Z 410.993,A -85,B 0,C 180,E1 -3664.834,E2 -3664.834} C_VEL
LIN {X 0,Y 545.226,Z 420.26,A -85,B 0,C 180,E1 -3667.652,E2 -3667.652} C_VEL
LIN {X 0,Y 545.077,Z 429.527,A -85,B 0,C 180,E1 -3670.415,E2 -3670.415} C_VEL
LIN {X 0,Y 544.952,Z 438.794,A -85,B 0,C 180,E1 -3673.134,E2 -3673.134} C_VEL
LIN {X 0,Y 544.857,Z 448.061,A -85,B 0,C 180,E1 -3675.815,E2 -3675.815} C_VEL
LIN {X 0,Y 544.804,Z 451.536,A -85,B 0,C 180,E1 -3676.812,E2 -3676.812} C_VEL
LIN {X 0,Y 546.174,Z 460.589,A -85,B 0,C 180,E1 -3677.035,E2 -3677.035} C_VEL
LIN {X 0,Y 546.018,Z 473.224,A -85,B 0,C 180,E1 -3677.41,E2 -3677.41} C_VEL
LIN {X 0,Y 545.789,Z 485.522,A -85,B 0,C 180,E1 -3677.923,E2 -3677.923} C_VEL
LIN {X 0,Y 545.59,Z 497.627,A -85,B 0,C 180,E1 -3678.597,E2 -3678.597} C_VEL
LIN {X 0,Y 545.418,Z 509.118,A -85,B 0,C 180,E1 -3679.421,E2 -3679.421} C_VEL
LIN {X 0,Y 545.164,Z 519.555,A -85,B 0,C 180,E1 -3680.354,E2 -3680.354} C_VEL
LIN {X 0,Y 545.028,Z 528.003,A -85,B 0,C 180,E1 -3681.287,E2 -3681.287} C_VEL
LIN {X 0,Y 544.858,Z 536.248,A -85,B 0,C 180,E1 -3682.404,E2 -3682.404} C_VEL
LIN {X 0,Y 544.732,Z 543.623,A -85,B 0,C 180,E1 -3683.656,E2 -3683.656} C_VEL
LIN {X 0,Y 544.653,Z 548.956,A -85,B 0,C 180,E1 -3684.819,E2 -3684.819} C_VEL
LIN {X 0,Y 544.683,Z 552.9,A -85,B 0,C 180,E1 -3685.932,E2 -3685.932} C_VEL
LIN {X 0,Y 544.65,Z 555.812,A -85,B 0,C 180,E1 -3687.043,E2 -3687.043} C_VEL
LIN {X 0,Y 544.546,Z 558.187,A -85,B 0,C 180,E1 -3688.522,E2 -3688.522} C_VEL
LIN {X 0,Y 544.541,Z 559,A -85,B 0,C 180,E1 -3690.001,E2 -3690.001} C_VEL
LIN {X 0,Y 544.546,Z 558.185,A -85,B 0,C 180,E1 -3691.48,E2 -3691.48} C_VEL
LIN {X 0,Y 544.651,Z 555.807,A -85,B 0,C 180,E1 -3692.96,E2 -3692.96} C_VEL
LIN {X 0,Y 544.684,Z 552.892,A -85,B 0,C 180,E1 -3694.071,E2 -3694.071} C_VEL
LIN {X 0,Y 544.654,Z 548.944,A -85,B 0,C 180,E1 -3695.184,E2 -3695.184} C_VEL
LIN {X 0,Y 544.737,Z 543.594,A -85,B 0,C 180,E1 -3696.349,E2 -3696.349} C_VEL
LIN {X 0,Y 544.861,Z 536.229,A -85,B 0,C 180,E1 -3697.599,E2 -3697.599} C_VEL
LIN {X 0,Y 545.027,Z 527.98,A -85,B 0,C 180,E1 -3698.716,E2 -3698.716} C_VEL
LIN {X 0,Y 545.166,Z 519.526,A -85,B 0,C 180,E1 -3699.649,E2 -3699.649} C_VEL
LIN {X 0,Y 545.4,Z 509.082,A -85,B 0,C 180,E1 -3700.582,E2 -3700.582} C_VEL
LIN {X 0,Y 545.62,Z 497.649,A -85,B 0,C 180,E1 -3701.401,E2 -3701.401} C_VEL
LIN {X 0,Y 545.762,Z 487.388,A -85,B 0,C 180,E1 -3701.986,E2 -3701.986} C_VEL
LIN {X 0,Y 545.972,Z 475.731,A -85,B 0,C 180,E1 -3702.5,E2 -3702.5} C_VEL
LIN {X 0,Y 546.14,Z 462.303,A -85,B 0,C 180,E1 -3702.921,E2 -3702.921} C_VEL
LIN {X 0,Y 545.929,Z 458.311,A -85,B 0,C 180,E1 -3703.021,E2 -3703.021} C_VEL
LIN {X 0,Y 544.806,Z 451.526,A -85,B 0,C 180,E1 -3703.19,E2 -3703.19} C_VEL
LIN {X 0,Y 544.94,Z 441.432,A -85,B 0,C 180,E1 -3706.099,E2 -3706.099} C_VEL
LIN {X 0,Y 545.073,Z 430.841,A -85,B 0,C 180,E1 -3709.196,E2 -3709.196} C_VEL
LIN {X 0,Y 545.218,Z 420.25,A -85,B 0,C 180,E1 -3712.351,E2 -3712.351} C_VEL
LIN {X 0,Y 545.357,Z 410.983,A -85,B 0,C 180,E1 -3715.169,E2 -3715.169} C_VEL
LIN {X 0,Y 545.552,Z 401.715,A -85,B 0,C 180,E1 -3718.049,E2 -3718.049} C_VEL
LIN {X 0,Y 545.706,Z 392.448,A -85,B 0,C 180,E1 -3721.008,E2 -3721.008} C_VEL
LIN {X 0,Y 545.941,Z 384.453,A -85,B 0,C 180,E1 -3723.612,E2 -3723.612} C_VEL
LIN {X 0,Y 545.945,Z 377.86,A -85,B 0,C 180,E1 -3725.805,E2 -3725.805} C_VEL
LIN {X 0,Y 545.058,Z 372.594,A -85,B 0,C 180,E1 -3727.769,E2 -3727.769} C_VEL
LIN {X 0,Y 545.086,Z 372.591,A -85,B 0,C 180,E1 -3730.473,E2 -3730.473} C_VEL
LIN {X 0,Y 545.084,Z 372.59,A -85,B 0,C 180,E1 -3733.107,E2 -3733.107} C_VEL
LIN {X 0,Y 545.054,Z 372.593,A -85,B 0,C 180,E1 -3736.227,E2 -3736.227} C_VEL
LIN {X 0,Y 545.086,Z 372.589,A -85,B 0,C 180,E1 -3738.886,E2 -3738.886} C_VEL
LIN {X 0,Y 545.056,Z 372.595,A -85,B 0,C 180,E1 -3741.763,E2 -3741.763} C_VEL
LIN {X 0,Y 545.041,Z 372.595,A -85,B 0,C 180,E1 -3744.532,E2 -3744.532} C_VEL
LIN {X 0,Y 545.07,Z 372.591,A -85,B 0,C 180,E1 -3747.211,E2 -3747.211} C_VEL
LIN {X 0,Y 545.068,Z 372.591,A -85,B 0,C 180,E1 -3749.811,E2 -3749.811} C_VEL
LIN {X 0,Y 545.082,Z 372.59,A -85,B 0,C 180,E1 -3752.344,E2 -3752.344} C_VEL
LIN {X 0,Y 545.122,Z 372.585,A -85,B 0,C 180,E1 -3754.82,E2 -3754.82} C_VEL
LIN {X 0,Y 545.042,Z 372.595,A -85,B 0,C 180,E1 -3757.242,E2 -3757.242} C_VEL
LIN {X 0,Y 545.125,Z 372.586,A -85,B 0,C 180,E1 -3760.415,E2 -3760.415} C_VEL
LIN {X 0,Y 545.076,Z 372.591,A -85,B 0,C 180,E1 -3763.521,E2 -3763.521} C_VEL
LIN {X 0,Y 545.099,Z 372.588,A -85,B 0,C 180,E1 -3765.82,E2 -3765.82} C_VEL
LIN {X 0,Y 545.121,Z 372.584,A -85,B 0,C 180,E1 -3768.849,E2 -3768.849} C_VEL
LIN {X 0,Y 545.134,Z 372.585,A -85,B 0,C 180,E1 -3771.847,E2 -3771.847} C_VEL
LIN {X 0,Y 545.205,Z 372.575,A -85,B 0,C 180,E1 -3774.823,E2 -3774.823} C_VEL
LIN {X 0,Y 545.199,Z 372.575,A -85,B 0,C 180,E1 -3777.784,E2 -3777.784} C_VEL
LIN {X 0,Y 545.214,Z 372.573,A -85,B 0,C 180,E1 -3780.739,E2 -3780.739} C_VEL
LIN {X 0,Y 545.175,Z 372.578,A -85,B 0,C 180,E1 -3782.956,E2 -3782.956} C_VEL
LIN {X 0,Y 545.173,Z 372.578,A -85,B 0,C 180,E1 -3785.919,E2 -3785.919} C_VEL
LIN {X 0,Y 545.124,Z 372.583,A -85,B 0,C 180,E1 -3788.9,E2 -3788.9} C_VEL
LIN {X 0,Y 545.139,Z 372.582,A -85,B 0,C 180,E1 -3791.904,E2 -3791.904} C_VEL
LIN {X 0,Y 545.089,Z 372.588,A -85,B 0,C 180,E1 -3794.943,E2 -3794.943} C_VEL
LIN {X 0,Y 545.08,Z 372.59,A -85,B 0,C 180,E1 -3798.026,E2 -3798.026} C_VEL
LIN {X 0,Y 545.096,Z 372.587,A -85,B 0,C 180,E1 -3800.372,E2 -3800.372} C_VEL
LIN {X 0,Y 545.085,Z 372.589,A -85,B 0,C 180,E1 -3803.559,E2 -3803.559} C_VEL
LIN {X 0,Y 545.082,Z 372.591,A -85,B 0,C 180,E1 -3806,E2 -3806} C_VEL
LIN {X 0,Y 545.093,Z 372.587,A -85,B 0,C 180,E1 -3808.748,E2 -3808.748} C_VEL
LIN {X 0,Y 545.062,Z 372.592,A -85,B 0,C 180,E1 -3811.679,E2 -3811.679} C_VEL
LIN {X 0,Y 545.066,Z 372.591,A -85,B 0,C 180,E1 -3814.564,E2 -3814.564} C_VEL
LIN {X 0,Y 545.065,Z 372.591,A -85,B 0,C 180,E1 -3817.007,E2 -3817.007} C_VEL
LIN {X 0,Y 544.357,Z 372.681,A -85,B 0,C 180,E1 -3817.624,E2 -3817.624} C_VEL
LIN {X 0,Y 541.491,Z 373.037,A -85,B 0,C 180,E1 -3818.625,E2 -3818.625} C_VEL
LIN {X 0,Y 539.104,Z 373.336,A -85,B 0,C 180,E1 -3819.43,E2 -3819.43} C_VEL
LIN {X 0,Y 538.095,Z 373.459,A -85,B 0,C 180,E1 -3820.052,E2 -3820.052} C_VEL
LIN {X 0,Y 538.02,Z 373.467,A -85,B 0,C 180,E1 -3820.263,E2 -3820.263} C_VEL
LIN {X 0,Y 538.031,Z 373.468,A -85,B 0,C 180,E1 -3822.987,E2 -3822.987} C_VEL
LIN {X 0,Y 538.007,Z 373.469,A -85,B 0,C 180,E1 -3826.184,E2 -3826.184} C_VEL
LIN {X 0,Y 538.054,Z 373.465,A -85,B 0,C 180,E1 -3829.252,E2 -3829.252} C_VEL
LIN {X 0,Y 537.998,Z 373.472,A -85,B 0,C 180,E1 -3832.122,E2 -3832.122} C_VEL
LIN {X 0,Y 538.004,Z 373.472,A -85,B 0,C 180,E1 -3834.915,E2 -3834.915} C_VEL
LIN {X 0,Y 538.024,Z 373.468,A -85,B 0,C 180,E1 -3837.617,E2 -3837.617} C_VEL
LIN {X 0,Y 538.02,Z 373.47,A -85,B 0,C 180,E1 -3840.238,E2 -3840.238} C_VEL
LIN {X 0,Y 538.06,Z 373.464,A -85,B 0,C 180,E1 -3842.795,E2 -3842.795} C_VEL
LIN {X 0,Y 538.054,Z 373.466,A -85,B 0,C 180,E1 -3845.292,E2 -3845.292} C_VEL
LIN {X 0,Y 538.028,Z 373.47,A -85,B 0,C 180,E1 -3848.545,E2 -3848.545} C_VEL
LIN {X 0,Y 538.039,Z 373.467,A -85,B 0,C 180,E1 -3850.939,E2 -3850.939} C_VEL
LIN {X 0,Y 538.022,Z 373.469,A -85,B 0,C 180,E1 -3853.298,E2 -3853.298} C_VEL
LIN {X 0,Y 538.07,Z 373.463,A -85,B 0,C 180,E1 -3855.63,E2 -3855.63} C_VEL
LIN {X 0,Y 537.981,Z 373.476,A -85,B 0,C 180,E1 -3858.457,E2 -3858.457} C_VEL
LIN {X 0,Y 537.844,Z 373.493,A -85,B 0,C 180,E1 -3859.458,E2 -3859.458} C_VEL
LIN {X 0,Y 537.771,Z 374.783,A -85,B 0,C 180,E1 -3860.976,E2 -3860.976} C_VEL
LIN {X 0,Y 537.736,Z 378.164,A -85,B 0,C 180,E1 -3863.997,E2 -3863.997} C_VEL
LIN {X 0,Y 537.721,Z 380.687,A -85,B 0,C 180,E1 -3866.252,E2 -3866.252} C_VEL
LIN {X 0,Y 537.606,Z 384.034,A -85,B 0,C 180,E1 -3869.25,E2 -3869.25} C_VEL
LIN {X 0,Y 537.541,Z 386.54,A -85,B 0,C 180,E1 -3871.497,E2 -3871.497} C_VEL
LIN {X 0,Y 537.607,Z 389.867,A -85,B 0,C 180,E1 -3874.497,E2 -3874.497} C_VEL
LIN {X 0,Y 537.546,Z 392.371,A -85,B 0,C 180,E1 -3876.756,E2 -3876.756} C_VEL
LIN {X 0,Y 537.484,Z 395.774,A -85,B 0,C 180,E1 -3879.738,E2 -3879.738} C_VEL
LIN {X 0,Y 539.179,Z 406.275,A -85,B 0,C 180,E1 -3880.062,E2 -3880.062} C_VEL
LIN {X 0,Y 539.032,Z 418.983,A -85,B 0,C 180,E1 -3880.516,E2 -3880.516} C_VEL
LIN {X 0,Y 538.72,Z 430.94,A -85,B 0,C 180,E1 -3881.093,E2 -3881.093} C_VEL
LIN {X 0,Y 538.501,Z 442.359,A -85,B 0,C 180,E1 -3881.811,E2 -3881.811} C_VEL
LIN {X 0,Y 538.283,Z 452.721,A -85,B 0,C 180,E1 -3882.631,E2 -3882.631} C_VEL
LIN {X 0,Y 538.034,Z 462.639,A -85,B 0,C 180,E1 -3883.597,E2 -3883.597} C_VEL
LIN {X 0,Y 537.881,Z 471.503,A -85,B 0,C 180,E1 -3884.665,E2 -3884.665} C_VEL
LIN {X 0,Y 537.762,Z 478.672,A -85,B 0,C 180,E1 -3885.733,E2 -3885.733} C_VEL
LIN {X 0,Y 537.651,Z 485.72,A -85,B 0,C 180,E1 -3887.051,E2 -3887.051} C_VEL
LIN {X 0,Y 537.548,Z 490.805,A -85,B 0,C 180,E1 -3888.285,E2 -3888.285} C_VEL
LIN {X 0,Y 537.51,Z 495.017,A -85,B 0,C 180,E1 -3889.71,E2 -3889.71} C_VEL
LIN {X 0,Y 537.464,Z 497.009,A -85,B 0,C 180,E1 -3890.672,E2 -3890.672} C_VEL
LIN {X 0,Y 537.473,Z 498.465,A -85,B 0,C 180,E1 -3891.814,E2 -3891.814} C_VEL
LIN {X 0,Y 537.465,Z 498.996,A -85,B 0,C 180,E1 -3893.095,E2 -3893.095} C_VEL
LIN {X 0,Y 537.48,Z 498.711,A -85,B 0,C 180,E1 -3893.911,E2 -3893.911} C_VEL
LIN {X 0,Y 537.455,Z 497.978,A -85,B 0,C 180,E1 -3894.734,E2 -3894.734} C_VEL
LIN {X 0,Y 537.474,Z 496.745,A -85,B 0,C 180,E1 -3895.561,E2 -3895.561} C_VEL
LIN {X 0,Y 537.526,Z 493.909,A -85,B 0,C 180,E1 -3896.811,E2 -3896.811} C_VEL
LIN {X 0,Y 537.565,Z 489.787,A -85,B 0,C 180,E1 -3898.075,E2 -3898.075} C_VEL
LIN {X 0,Y 537.669,Z 484.228,A -85,B 0,C 180,E1 -3899.35,E2 -3899.35} C_VEL
LIN {X 0,Y 537.807,Z 476.917,A -85,B 0,C 180,E1 -3900.638,E2 -3900.638} C_VEL
LIN {X 0,Y 537.916,Z 469.44,A -85,B 0,C 180,E1 -3901.691,E2 -3901.691} C_VEL
LIN {X 0,Y 538.144,Z 460.632,A -85,B 0,C 180,E1 -3902.705,E2 -3902.705} C_VEL
LIN {X 0,Y 538.335,Z 451.304,A -85,B 0,C 180,E1 -3903.584,E2 -3903.584} C_VEL
LIN {X 0,Y 538.602,Z 440.26,A -85,B 0,C 180,E1 -3904.422,E2 -3904.422} C_VEL
LIN {X 0,Y 538.809,Z 428.35,A -85,B 0,C 180,E1 -3905.135,E2 -3905.135} C_VEL
LIN {X 0,Y 539.017,Z 416.172,A -85,B 0,C 180,E1 -3905.693,E2 -3905.693} C_VEL
LIN {X 0,Y 538.982,Z 404.393,A -85,B 0,C 180,E1 -3906.087,E2 -3906.087} C_VEL
LIN {X 0,Y 537.484,Z 395.811,A -85,B 0,C 180,E1 -3906.349,E2 -3906.349} C_VEL
LIN {X 0,Y 537.491,Z 392.285,A -85,B 0,C 180,E1 -3909.515,E2 -3909.515} C_VEL
LIN {X 0,Y 537.552,Z 389.802,A -85,B 0,C 180,E1 -3911.822,E2 -3911.822} C_VEL
LIN {X 0,Y 537.616,Z 386.365,A -85,B 0,C 180,E1 -3914.9,E2 -3914.9} C_VEL
LIN {X 0,Y 537.668,Z 383.869,A -85,B 0,C 180,E1 -3917.179,E2 -3917.179} C_VEL
LIN {X 0,Y 537.653,Z 380.59,A -85,B 0,C 180,E1 -3920.17,E2 -3920.17} C_VEL
LIN {X 0,Y 537.736,Z 377.41,A -85,B 0,C 180,E1 -3923.044,E2 -3923.044} C_VEL
LIN {X 0,Y 537.76,Z 374.306,A -85,B 0,C 180,E1 -3925.808,E2 -3925.808} C_VEL
LIN {X 0,Y 537.811,Z 373.498,A -85,B 0,C 180,E1 -3926.751,E2 -3926.751} C_VEL
LIN {X 0,Y 538.017,Z 373.472,A -85,B 0,C 180,E1 -3929.553,E2 -3929.553} C_VEL
LIN {X 0,Y 538.031,Z 373.466,A -85,B 0,C 180,E1 -3931.95,E2 -3931.95} C_VEL
LIN {X 0,Y 538.057,Z 373.463,A -85,B 0,C 180,E1 -3934.466,E2 -3934.466} C_VEL
LIN {X 0,Y 538.04,Z 373.465,A -85,B 0,C 180,E1 -3936.929,E2 -3936.929} C_VEL
LIN {X 0,Y 538.059,Z 373.463,A -85,B 0,C 180,E1 -3940.147,E2 -3940.147} C_VEL
LIN {X 0,Y 538.007,Z 373.471,A -85,B 0,C 180,E1 -3943.298,E2 -3943.298} C_VEL
LIN {X 0,Y 538.045,Z 373.465,A -85,B 0,C 180,E1 -3945.63,E2 -3945.63} C_VEL
LIN {X 0,Y 538.071,Z 373.463,A -85,B 0,C 180,E1 -3948.701,E2 -3948.701} C_VEL
LIN {X 0,Y 538.072,Z 373.461,A -85,B 0,C 180,E1 -3951.739,E2 -3951.739} C_VEL
LIN {X 0,Y 538.173,Z 373.448,A -85,B 0,C 180,E1 -3954.755,E2 -3954.755} C_VEL
LIN {X 0,Y 538.156,Z 373.451,A -85,B 0,C 180,E1 -3957.755,E2 -3957.755} C_VEL
LIN {X 0,Y 538.169,Z 373.452,A -85,B 0,C 180,E1 -3960.748,E2 -3960.748} C_VEL
LIN {X 0,Y 538.128,Z 373.454,A -85,B 0,C 180,E1 -3962.995,E2 -3962.995} C_VEL
LIN {X 0,Y 538.107,Z 373.458,A -85,B 0,C 180,E1 -3965.998,E2 -3965.998} C_VEL
LIN {X 0,Y 538.053,Z 373.466,A -85,B 0,C 180,E1 -3969.018,E2 -3969.018} C_VEL
LIN {X 0,Y 538.063,Z 373.462,A -85,B 0,C 180,E1 -3972.063,E2 -3972.063} C_VEL
LIN {X 0,Y 538.026,Z 373.467,A -85,B 0,C 180,E1 -3975.144,E2 -3975.144} C_VEL
LIN {X 0,Y 538.019,Z 373.471,A -85,B 0,C 180,E1 -3978.271,E2 -3978.271} C_VEL
LIN {X 0,Y 538.025,Z 373.467,A -85,B 0,C 180,E1 -3980.652,E2 -3980.652} C_VEL
LIN {X 0,Y 538.042,Z 373.465,A -85,B 0,C 180,E1 -3983.071,E2 -3983.071} C_VEL
LIN {X 0,Y 538.03,Z 373.467,A -85,B 0,C 180,E1 -3985.675,E2 -3985.675} C_VEL
LIN {X 0,Y 538.031,Z 373.468,A -85,B 0,C 180,E1 -3988.051,E2 -3988.051} C_VEL
LIN {X 0,Y 538.003,Z 373.473,A -85,B 0,C 180,E1 -3990.628,E2 -3990.628} C_VEL
LIN {X 0,Y 538.028,Z 373.47,A -85,B 0,C 180,E1 -3993.284,E2 -3993.284} C_VEL
LIN {X 0,Y 538.014,Z 373.471,A -85,B 0,C 180,E1 -3996.003,E2 -3996.003} C_VEL
LIN {X 0,Y 537.998,Z 373.473,A -85,B 0,C 180,E1 -3998.832,E2 -3998.832} C_VEL
LIN {X 0,Y 538.045,Z 373.466,A -85,B 0,C 180,E1 -4001.772,E2 -4001.772} C_VEL
LIN {X 0,Y 538.02,Z 373.472,A -85,B 0,C 180,E1 -4005.142,E2 -4005.142} C_VEL
LIN {X 0,Y 538.033,Z 373.47,A -85,B 0,C 180,E1 -4008.23,E2 -4008.23} C_VEL
LIN {X 0,Y 538.05,Z 373.466,A -85,B 0,C 180,E1 -4010.413,E2 -4010.413} C_VEL
LIN {X 0,Y 538.025,Z 373.477,A -85,B 0,C 180,E1 -4011.999,E2 -4011.999} C_VEL
LIN {X 0,Y 538.991,Z 379.051,A -85,B 0,C 180,E1 -4014.075,E2 -4014.075} C_VEL
LIN {X 0,Y 538.945,Z 386.515,A -85,B 0,C 180,E1 -4016.572,E2 -4016.572} C_VEL
LIN {X 0,Y 538.715,Z 393.782,A -85,B 0,C 180,E1 -4018.984,E2 -4018.984} C_VEL
LIN {X 0,Y 538.553,Z 403.049,A -85,B 0,C 180,E1 -4021.981,E2 -4021.981} C_VEL
LIN {X 0,Y 538.326,Z 412.317,A -85,B 0,C 180,E1 -4024.896,E2 -4024.896} C_VEL
LIN {X 0,Y 538.203,Z 421.584,A -85,B 0,C 180,E1 -4027.749,E2 -4027.749} C_VEL
LIN {X 0,Y 538.02,Z 430.851,A -85,B 0,C 180,E1 -4030.545,E2 -4030.545} C_VEL
LIN {X 0,Y 537.892,Z 440.118,A -85,B 0,C 180,E1 -4033.297,E2 -4033.297} C_VEL
LIN {X 0,Y 537.789,Z 449.385,A -85,B 0,C 180,E1 -4036.011,E2 -4036.011} C_VEL
LIN {X 0,Y 537.746,Z 451.578,A -85,B 0,C 180,E1 -4036.648,E2 -4036.648} C_VEL
LIN {X 0,Y 539.249,Z 461.504,A -85,B 0,C 180,E1 -4036.89,E2 -4036.89} C_VEL
LIN {X 0,Y 539.096,Z 474.521,A -85,B 0,C 180,E1 -4037.293,E2 -4037.293} C_VEL
LIN {X 0,Y 538.851,Z 485.522,A -85,B 0,C 180,E1 -4037.766,E2 -4037.766} C_VEL
LIN {X 0,Y 538.639,Z 496.567,A -85,B 0,C 180,E1 -4038.38,E2 -4038.38} C_VEL
LIN {X 0,Y 538.419,Z 507.946,A -85,B 0,C 180,E1 -4039.187,E2 -4039.187} C_VEL
LIN {X 0,Y 538.2,Z 517.619,A -85,B 0,C 180,E1 -4040.038,E2 -4040.038} C_VEL
LIN {X 0,Y 538.014,Z 526.427,A -85,B 0,C 180,E1 -4040.983,E2 -4040.983} C_VEL
LIN {X 0,Y 537.828,Z 535.012,A -85,B 0,C 180,E1 -4042.115,E2 -4042.115} C_VEL
LIN {X 0,Y 537.704,Z 541.876,A -85,B 0,C 180,E1 -4043.246,E2 -4043.246} C_VEL
LIN {X 0,Y 537.676,Z 547.372,A -85,B 0,C 180,E1 -4044.376,E2 -4044.376} C_VEL
LIN {X 0,Y 537.557,Z 551.682,A -85,B 0,C 180,E1 -4045.502,E2 -4045.502} C_VEL
LIN {X 0,Y 537.591,Z 553.962,A -85,B 0,C 180,E1 -4046.254,E2 -4046.254} C_VEL
LIN {X 0,Y 537.551,Z 555.811,A -85,B 0,C 180,E1 -4047.004,E2 -4047.004} C_VEL
LIN {X 0,Y 537.49,Z 557.2,A -85,B 0,C 180,E1 -4047.753,E2 -4047.753} C_VEL
LIN {X 0,Y 537.442,Z 558.786,A -85,B 0,C 180,E1 -4049.252,E2 -4049.252} C_VEL
LIN {X 0,Y 537.442,Z 559,A -85,B 0,C 180,E1 -4050.001,E2 -4050.001} C_VEL
LIN {X 0,Y 537.451,Z 558.185,A -85,B 0,C 180,E1 -4051.5,E2 -4051.5} C_VEL
LIN {X 0,Y 537.49,Z 557.197,A -85,B 0,C 180,E1 -4052.249,E2 -4052.249} C_VEL
LIN {X 0,Y 537.551,Z 555.807,A -85,B 0,C 180,E1 -4052.999,E2 -4052.999} C_VEL
LIN {X 0,Y 537.604,Z 552.892,A -85,B 0,C 180,E1 -4054.125,E2 -4054.125} C_VEL
LIN {X 0,Y 537.588,Z 548.944,A -85,B 0,C 180,E1 -4055.252,E2 -4055.252} C_VEL
LIN {X 0,Y 537.652,Z 544.087,A -85,B 0,C 180,E1 -4056.334,E2 -4056.334} C_VEL
LIN {X 0,Y 537.792,Z 537.46,A -85,B 0,C 180,E1 -4057.51,E2 -4057.51} C_VEL
LIN {X 0,Y 537.971,Z 529.468,A -85,B 0,C 180,E1 -4058.642,E2 -4058.642} C_VEL
LIN {X 0,Y 538.12,Z 521.324,A -85,B 0,C 180,E1 -4059.587,E2 -4059.587} C_VEL
LIN {X 0,Y 538.343,Z 511.387,A -85,B 0,C 180,E1 -4060.532,E2 -4060.532} C_VEL
LIN {X 0,Y 538.557,Z 501.569,A -85,B 0,C 180,E1 -4061.289,E2 -4061.289} C_VEL
LIN {X 0,Y 538.743,Z 490.594,A -85,B 0,C 180,E1 -4061.97,E2 -4061.97} C_VEL
LIN {X 0,Y 538.988,Z 478.081,A -85,B 0,C 180,E1 -4062.569,E2 -4062.569} C_VEL
LIN {X 0,Y 539.188,Z 465.045,A -85,B 0,C 180,E1 -4063.019,E2 -4063.019} C_VEL
LIN {X 0,Y 539.027,Z 459.45,A -85,B 0,C 180,E1 -4063.167,E2 -4063.167} C_VEL
LIN {X 0,Y 537.739,Z 451.526,A -85,B 0,C 180,E1 -4063.367,E2 -4063.367} C_VEL
LIN {X 0,Y 537.88,Z 441.432,A -85,B 0,C 180,E1 -4066.316,E2 -4066.316} C_VEL
LIN {X 0,Y 538.002,Z 432.164,A -85,B 0,C 180,E1 -4069.062,E2 -4069.062} C_VEL
LIN {X 0,Y 538.18,Z 422.406,A -85,B 0,C 180,E1 -4072.001,E2 -4072.001} C_VEL
LIN {X 0,Y 538.333,Z 412.306,A -85,B 0,C 180,E1 -4075.107,E2 -4075.107} C_VEL
LIN {X 0,Y 538.54,Z 403.039,A -85,B 0,C 180,E1 -4078.023,E2 -4078.023} C_VEL
LIN {X 0,Y 538.724,Z 393.772,A -85,B 0,C 180,E1 -4081.019,E2 -4081.019} C_VEL
LIN {X 0,Y 538.969,Z 385.517,A -85,B 0,C 180,E1 -4083.722,E2 -4083.722} C_VEL
LIN {X 0,Y 538.959,Z 378.976,A -85,B 0,C 180,E1 -4085.931,E2 -4085.931} C_VEL
LIN {X 0,Y 538.017,Z 373.471,A -85,B 0,C 180,E1 -4088.037,E2 -4088.037} C_VEL
LIN {X 0,Y 538.054,Z 373.465,A -85,B 0,C 180,E1 -4090.776,E2 -4090.776} C_VEL
LIN {X 0,Y 538.008,Z 373.47,A -85,B 0,C 180,E1 -4093.816,E2 -4093.816} C_VEL
LIN {X 0,Y 538.031,Z 373.468,A -85,B 0,C 180,E1 -4097.013,E2 -4097.013} C_VEL
LIN {X 0,Y 538.053,Z 373.465,A -85,B 0,C 180,E1 -4099.253,E2 -4099.253} C_VEL
LIN {X 0,Y 537.996,Z 373.472,A -85,B 0,C 180,E1 -4102.122,E2 -4102.122} C_VEL
LIN {X 0,Y 538.002,Z 373.473,A -85,B 0,C 180,E1 -4104.916,E2 -4104.916} C_VEL
LIN {X 0,Y 538.021,Z 373.468,A -85,B 0,C 180,E1 -4107.617,E2 -4107.617} C_VEL
LIN {X 0,Y 538.021,Z 373.47,A -85,B 0,C 180,E1 -4110.239,E2 -4110.239} C_VEL
LIN {X 0,Y 538.059,Z 373.465,A -85,B 0,C 180,E1 -4112.796,E2 -4112.796} C_VEL
LIN {X 0,Y 538.052,Z 373.465,A -85,B 0,C 180,E1 -4115.293,E2 -4115.293} C_VEL
LIN {X 0,Y 538.027,Z 373.469,A -85,B 0,C 180,E1 -4118.546,E2 -4118.546} C_VEL
LIN {X 0,Y 538.041,Z 373.466,A -85,B 0,C 180,E1 -4120.94,E2 -4120.94} C_VEL
LIN {X 0,Y 538.028,Z 373.469,A -85,B 0,C 180,E1 -4123.299,E2 -4123.299} C_VEL
LIN {X 0,Y 538.068,Z 373.464,A -85,B 0,C 180,E1 -4125.631,E2 -4125.631} C_VEL
LIN {X 0,Y 538.081,Z 373.463,A -85,B 0,C 180,E1 -4128.702,E2 -4128.702} C_VEL
LIN {X 0,Y 538.091,Z 373.461,A -85,B 0,C 180,E1 -4131.74,E2 -4131.74} C_VEL
LIN {X 0,Y 538.162,Z 373.453,A -85,B 0,C 180,E1 -4134.755,E2 -4134.755} C_VEL
LIN {X 0,Y 538.171,Z 373.45,A -85,B 0,C 180,E1 -4137.755,E2 -4137.755} C_VEL
LIN {X 0,Y 538.184,Z 373.448,A -85,B 0,C 180,E1 -4140.748,E2 -4140.748} C_VEL
LIN {X 0,Y 538.141,Z 373.454,A -85,B 0,C 180,E1 -4142.994,E2 -4142.994} C_VEL
LIN {X 0,Y 538.124,Z 373.457,A -85,B 0,C 180,E1 -4145.997,E2 -4145.997} C_VEL
LIN {X 0,Y 538.075,Z 373.461,A -85,B 0,C 180,E1 -4149.017,E2 -4149.017} C_VEL
LIN {X 0,Y 538.087,Z 373.461,A -85,B 0,C 180,E1 -4152.062,E2 -4152.062} C_VEL
LIN {X 0,Y 538.049,Z 373.465,A -85,B 0,C 180,E1 -4155.144,E2 -4155.144} C_VEL
LIN {X 0,Y 538.032,Z 373.467,A -85,B 0,C 180,E1 -4158.27,E2 -4158.27} C_VEL
LIN {X 0,Y 538.041,Z 373.467,A -85,B 0,C 180,E1 -4160.651,E2 -4160.651} C_VEL
LIN {X 0,Y 538.008,Z 373.472,A -85,B 0,C 180,E1 -4163.888,E2 -4163.888} C_VEL
LIN {X 0,Y 538.045,Z 373.465,A -85,B 0,C 180,E1 -4166.367,E2 -4166.367} C_VEL
LIN {X 0,Y 538.035,Z 373.467,A -85,B 0,C 180,E1 -4168.933,E2 -4168.933} C_VEL
LIN {X 0,Y 538.014,Z 373.47,A -85,B 0,C 180,E1 -4171.887,E2 -4171.887} C_VEL
LIN {X 0,Y 538.016,Z 373.469,A -85,B 0,C 180,E1 -4174.617,E2 -4174.617} C_VEL
LIN {X 0,Y 538.008,Z 373.471,A -85,B 0,C 180,E1 -4177.169,E2 -4177.169} C_VEL
LIN {X 0,Y 538.02,Z 373.467,A -85,B 0,C 180,E1 -4180.263,E2 -4180.263} C_VEL
LIN {X 0,Y 537.372,Z 373.551,A -85,B 0,C 180,E1 -4180.888,E2 -4180.888} C_VEL
LIN {X 0,Y 534.52,Z 373.91,A -85,B 0,C 180,E1 -4181.903,E2 -4181.903} C_VEL
LIN {X 0,Y 532.094,Z 374.213,A -85,B 0,C 180,E1 -4182.72,E2 -4182.72} C_VEL
LIN {X 0,Y 531.044,Z 374.341,A -85,B 0,C 180,E1 -4183.351,E2 -4183.351} C_VEL
LIN {X 0,Y 530.956,Z 374.35,A -85,B 0,C 180,E1 -4183.565,E2 -4183.565} C_VEL
LIN {X 0,Y 530.959,Z 374.348,A -85,B 0,C 180,E1 -4186.504,E2 -4186.504} C_VEL
LIN {X 0,Y 530.991,Z 374.346,A -85,B 0,C 180,E1 -4188.976,E2 -4188.976} C_VEL
LIN {X 0,Y 530.963,Z 374.348,A -85,B 0,C 180,E1 -4191.529,E2 -4191.529} C_VEL
LIN {X 0,Y 530.96,Z 374.348,A -85,B 0,C 180,E1 -4194.379,E2 -4194.379} C_VEL
LIN {X 0,Y 530.972,Z 374.348,A -85,B 0,C 180,E1 -4197.133,E2 -4197.133} C_VEL
LIN {X 0,Y 530.967,Z 374.347,A -85,B 0,C 180,E1 -4199.802,E2 -4199.802} C_VEL
LIN {X 0,Y 531.017,Z 374.342,A -85,B 0,C 180,E1 -4202.467,E2 -4202.467} C_VEL
LIN {X 0,Y 531.011,Z 374.342,A -85,B 0,C 180,E1 -4204.942,E2 -4204.942} C_VEL
LIN {X 0,Y 530.977,Z 374.346,A -85,B 0,C 180,E1 -4208.246,E2 -4208.246} C_VEL
LIN {X 0,Y 530.998,Z 374.345,A -85,B 0,C 180,E1 -4210.676,E2 -4210.676} C_VEL
LIN {X 0,Y 530.986,Z 374.345,A -85,B 0,C 180,E1 -4213.07,E2 -4213.07} C_VEL
LIN {X 0,Y 531.025,Z 374.34,A -85,B 0,C 180,E1 -4215.435,E2 -4215.435} C_VEL
LIN {X 0,Y 530.932,Z 374.354,A -85,B 0,C 180,E1 -4218.546,E2 -4218.546} C_VEL
LIN {X 0,Y 530.688,Z 374.482,A -85,B 0,C 180,E1 -4220.085,E2 -4220.085} C_VEL
LIN {X 0,Y 530.688,Z 377.033,A -85,B 0,C 180,E1 -4222.389,E2 -4222.389} C_VEL
LIN {X 0,Y 530.672,Z 380.425,A -85,B 0,C 180,E1 -4225.441,E2 -4225.441} C_VEL
LIN {X 0,Y 530.533,Z 383.833,A -85,B 0,C 180,E1 -4228.48,E2 -4228.48} C_VEL
LIN {X 0,Y 530.485,Z 386.347,A -85,B 0,C 180,E1 -4230.758,E2 -4230.758} C_VEL
LIN {X 0,Y 530.574,Z 389.701,A -85,B 0,C 180,E1 -4233.796,E2 -4233.796} C_VEL
LIN {X 0,Y 530.53,Z 392.67,A -85,B 0,C 180,E1 -4236.518,E2 -4236.518} C_VEL
LIN {X 0,Y 530.418,Z 396.177,A -85,B 0,C 180,E1 -4239.58,E2 -4239.58} C_VEL
LIN {X 0,Y 532.268,Z 407.147,A -85,B 0,C 180,E1 -4239.906,E2 -4239.906} C_VEL
LIN {X 0,Y 532.094,Z 419.712,A -85,B 0,C 180,E1 -4240.366,E2 -4240.366} C_VEL
LIN {X 0,Y 531.774,Z 431.541,A -85,B 0,C 180,E1 -4240.95,E2 -4240.95} C_VEL
LIN {X 0,Y 531.567,Z 442.181,A -85,B 0,C 180,E1 -4241.63,E2 -4241.63} C_VEL
LIN {X 0,Y 531.322,Z 452.01,A -85,B 0,C 180,E1 -4242.411,E2 -4242.411} C_VEL
LIN {X 0,Y 531.047,Z 462.004,A -85,B 0,C 180,E1 -4243.389,E2 -4243.389} C_VEL
LIN {X 0,Y 530.859,Z 470.178,A -85,B 0,C 180,E1 -4244.371,E2 -4244.371} C_VEL
LIN {X 0,Y 530.706,Z 478.195,A -85,B 0,C 180,E1 -4245.553,E2 -4245.553} C_VEL
LIN {X 0,Y 530.602,Z 483.683,A -85,B 0,C 180,E1 -4246.544,E2 -4246.544} C_VEL
LIN {X 0,Y 530.503,Z 489.001,A -85,B 0,C 180,E1 -4247.738,E2 -4247.738} C_VEL
LIN {X 0,Y 530.459,Z 493.1,A -85,B 0,C 180,E1 -4248.939,E2 -4248.939} C_VEL
LIN {X 0,Y 530.366,Z 496.092,A -85,B 0,C 180,E1 -4250.151,E2 -4250.151} C_VEL
LIN {X 0,Y 530.353,Z 497.485,A -85,B 0,C 180,E1 -4250.963,E2 -4250.963} C_VEL
LIN {X 0,Y 530.374,Z 498.568,A -85,B 0,C 180,E1 -4251.94,E2 -4251.94} C_VEL
LIN {X 0,Y 530.392,Z 498.927,A -85,B 0,C 180,E1 -4253.421,E2 -4253.421} C_VEL
LIN {X 0,Y 530.358,Z 498.498,A -85,B 0,C 180,E1 -4254.253,E2 -4254.253} C_VEL
LIN {X 0,Y 530.382,Z 496.539,A -85,B 0,C 180,E1 -4255.703,E2 -4255.703} C_VEL
LIN {X 0,Y 530.428,Z 494.155,A -85,B 0,C 180,E1 -4256.773,E2 -4256.773} C_VEL
LIN {X 0,Y 530.478,Z 490.12,A -85,B 0,C 180,E1 -4258.053,E2 -4258.053} C_VEL
LIN {X 0,Y 530.6,Z 484.656,A -85,B 0,C 180,E1 -4259.343,E2 -4259.343} C_VEL
LIN {X 0,Y 530.713,Z 477.83,A -85,B 0,C 180,E1 -4260.597,E2 -4260.597} C_VEL
LIN {X 0,Y 530.865,Z 469.949,A -85,B 0,C 180,E1 -4261.749,E2 -4261.749} C_VEL
LIN {X 0,Y 531.123,Z 460.596,A -85,B 0,C 180,E1 -4262.853,E2 -4262.853} C_VEL
LIN {X 0,Y 531.363,Z 451.308,A -85,B 0,C 180,E1 -4263.743,E2 -4263.743} C_VEL
LIN {X 0,Y 531.623,Z 441.248,A -85,B 0,C 180,E1 -4264.525,E2 -4264.525} C_VEL
LIN {X 0,Y 531.871,Z 429.145,A -85,B 0,C 180,E1 -4265.271,E2 -4265.271} C_VEL
LIN {X 0,Y 532.113,Z 417.508,A -85,B 0,C 180,E1 -4265.82,E2 -4265.82} C_VEL
LIN {X 0,Y 532.103,Z 405.356,A -85,B 0,C 180,E1 -4266.244,E2 -4266.244} C_VEL
LIN {X 0,Y 530.392,Z 396.214,A -85,B 0,C 180,E1 -4266.511,E2 -4266.511} C_VEL
LIN {X 0,Y 530.417,Z 392.94,A -85,B 0,C 180,E1 -4269.491,E2 -4269.491} C_VEL
LIN {X 0,Y 530.477,Z 390.134,A -85,B 0,C 180,E1 -4272.105,E2 -4272.105} C_VEL
LIN {X 0,Y 530.535,Z 387.368,A -85,B 0,C 180,E1 -4274.592,E2 -4274.592} C_VEL
LIN {X 0,Y 530.577,Z 384.183,A -85,B 0,C 180,E1 -4277.504,E2 -4277.504} C_VEL
LIN {X 0,Y 530.591,Z 381.256,A -85,B 0,C 180,E1 -4280.193,E2 -4280.193} C_VEL
LIN {X 0,Y 530.657,Z 377.674,A -85,B 0,C 180,E1 -4283.418,E2 -4283.418} C_VEL
LIN {X 0,Y 530.695,Z 374.594,A -85,B 0,C 180,E1 -4286.206,E2 -4286.206} C_VEL
LIN {X 0,Y 530.883,Z 374.361,A -85,B 0,C 180,E1 -4288.026,E2 -4288.026} C_VEL
LIN {X 0,Y 530.989,Z 374.346,A -85,B 0,C 180,E1 -4290.869,E2 -4290.869} C_VEL
LIN {X 0,Y 530.994,Z 374.343,A -85,B 0,C 180,E1 -4293.256,E2 -4293.256} C_VEL
LIN {X 0,Y 530.998,Z 374.343,A -85,B 0,C 180,E1 -4295.952,E2 -4295.952} C_VEL
LIN {X 0,Y 530.988,Z 374.347,A -85,B 0,C 180,E1 -4299.062,E2 -4299.062} C_VEL
LIN {X 0,Y 530.996,Z 374.342,A -85,B 0,C 180,E1 -4302.277,E2 -4302.277} C_VEL
LIN {X 0,Y 530.999,Z 374.342,A -85,B 0,C 180,E1 -4305.435,E2 -4305.435} C_VEL
LIN {X 0,Y 531.028,Z 374.342,A -85,B 0,C 180,E1 -4308.55,E2 -4308.55} C_VEL
LIN {X 0,Y 531.041,Z 374.337,A -85,B 0,C 180,E1 -4311.629,E2 -4311.629} C_VEL
LIN {X 0,Y 531.128,Z 374.325,A -85,B 0,C 180,E1 -4314.685,E2 -4314.685} C_VEL
LIN {X 0,Y 531.127,Z 374.327,A -85,B 0,C 180,E1 -4317.725,E2 -4317.725} C_VEL
LIN {X 0,Y 531.138,Z 374.328,A -85,B 0,C 180,E1 -4320.758,E2 -4320.758} C_VEL
LIN {X 0,Y 531.094,Z 374.33,A -85,B 0,C 180,E1 -4323.034,E2 -4323.034} C_VEL
LIN {X 0,Y 531.066,Z 374.336,A -85,B 0,C 180,E1 -4326.077,E2 -4326.077} C_VEL
LIN {X 0,Y 531.013,Z 374.341,A -85,B 0,C 180,E1 -4329.139,E2 -4329.139} C_VEL
LIN {X 0,Y 531.038,Z 374.34,A -85,B 0,C 180,E1 -4331.677,E2 -4331.677} C_VEL
LIN {X 0,Y 531.009,Z 374.34,A -85,B 0,C 180,E1 -4334.957,E2 -4334.957} C_VEL
LIN {X 0,Y 530.997,Z 374.342,A -85,B 0,C 180,E1 -4337.723,E2 -4337.723} C_VEL
LIN {X 0,Y 530.989,Z 374.346,A -85,B 0,C 180,E1 -4340.938,E2 -4340.938} C_VEL
LIN {X 0,Y 531.009,Z 374.343,A -85,B 0,C 180,E1 -4344.051,E2 -4344.051} C_VEL
LIN {X 0,Y 530.994,Z 374.345,A -85,B 0,C 180,E1 -4346.744,E2 -4346.744} C_VEL
LIN {X 0,Y 530.965,Z 374.349,A -85,B 0,C 180,E1 -4349.324,E2 -4349.324} C_VEL
LIN {X 0,Y 530.964,Z 374.348,A -85,B 0,C 180,E1 -4352.105,E2 -4352.105} C_VEL
LIN {X 0,Y 530.973,Z 374.347,A -85,B 0,C 180,E1 -4354.856,E2 -4354.856} C_VEL
LIN {X 0,Y 530.958,Z 374.349,A -85,B 0,C 180,E1 -4357.509,E2 -4357.509} C_VEL
LIN {X 0,Y 530.995,Z 374.344,A -85,B 0,C 180,E1 -4360.432,E2 -4360.432} C_VEL
LIN {X 0,Y 530.951,Z 374.351,A -85,B 0,C 180,E1 -4363.496,E2 -4363.496} C_VEL
LIN {X 0,Y 530.954,Z 374.353,A -85,B 0,C 180,E1 -4366.507,E2 -4366.507} C_VEL
LIN {X 0,Y 531.017,Z 374.343,A -85,B 0,C 180,E1 -4369.573,E2 -4369.573} C_VEL
LIN {X 0,Y 530.97,Z 374.467,A -85,B 0,C 180,E1 -4371.775,E2 -4371.775} C_VEL
LIN {X 0,Y 532.014,Z 380.454,A -85,B 0,C 180,E1 -4374.09,E2 -4374.09} C_VEL
LIN {X 0,Y 532.003,Z 387.139,A -85,B 0,C 180,E1 -4376.332,E2 -4376.332} C_VEL
LIN {X 0,Y 531.755,Z 395.825,A -85,B 0,C 180,E1 -4379.214,E2 -4379.214} C_VEL
LIN {X 0,Y 531.486,Z 405.503,A -85,B 0,C 180,E1 -4382.371,E2 -4382.371} C_VEL
LIN {X 0,Y 531.319,Z 413.64,A -85,B 0,C 180,E1 -4384.96,E2 -4384.96} C_VEL
LIN {X 0,Y 531.158,Z 422.917,A -85,B 0,C 180,E1 -4387.851,E2 -4387.851} C_VEL
LIN {X 0,Y 530.963,Z 432.175,A -85,B 0,C 180,E1 -4390.678,E2 -4390.678} C_VEL
LIN {X 0,Y 530.823,Z 441.442,A -85,B 0,C 180,E1 -4393.464,E2 -4393.464} C_VEL
LIN {X 0,Y 530.707,Z 451.371,A -85,B 0,C 180,E1 -4396.407,E2 -4396.407} C_VEL
LIN {X 0,Y 530.707,Z 451.841,A -85,B 0,C 180,E1 -4396.474,E2 -4396.474} C_VEL
LIN {X 0,Y 532.347,Z 462.419,A -85,B 0,C 180,E1 -4396.741,E2 -4396.741} C_VEL
LIN {X 0,Y 532.172,Z 474.522,A -85,B 0,C 180,E1 -4397.125,E2 -4397.125} C_VEL
LIN {X 0,Y 531.913,Z 485.523,A -85,B 0,C 180,E1 -4397.603,E2 -4397.603} C_VEL
LIN {X 0,Y 531.652,Z 497.246,A -85,B 0,C 180,E1 -4398.268,E2 -4398.268} C_VEL
LIN {X 0,Y 531.445,Z 507.945,A -85,B 0,C 180,E1 -4399.043,E2 -4399.043} C_VEL
LIN {X 0,Y 531.194,Z 517.618,A -85,B 0,C 180,E1 -4399.905,E2 -4399.905} C_VEL
LIN {X 0,Y 530.968,Z 526.427,A -85,B 0,C 180,E1 -4400.862,E2 -4400.862} C_VEL
LIN {X 0,Y 530.778,Z 535.012,A -85,B 0,C 180,E1 -4402.01,E2 -4402.01} C_VEL
LIN {X 0,Y 530.635,Z 541.877,A -85,B 0,C 180,E1 -4403.156,E2 -4403.156} C_VEL
LIN {X 0,Y 530.61,Z 547.372,A -85,B 0,C 180,E1 -4404.301,E2 -4404.301} C_VEL
LIN {X 0,Y 530.457,Z 551.682,A -85,B 0,C 180,E1 -4405.442,E2 -4405.442} C_VEL
LIN {X 0,Y 530.516,Z 553.962,A -85,B 0,C 180,E1 -4406.204,E2 -4406.204} C_VEL
LIN {X 0,Y 530.457,Z 555.811,A -85,B 0,C 180,E1 -4406.964,E2 -4406.964} C_VEL
LIN {X 0,Y 530.411,Z 557.2,A -85,B 0,C 180,E1 -4407.723,E2 -4407.723} C_VEL
LIN {X 0,Y 530.344,Z 558.786,A -85,B 0,C 180,E1 -4409.242,E2 -4409.242} C_VEL
LIN {X 0,Y 530.342,Z 559,A -85,B 0,C 180,E1 -4410.001,E2 -4410.001} C_VEL
LIN {X 0,Y 530.361,Z 558.185,A -85,B 0,C 180,E1 -4411.52,E2 -4411.52} C_VEL
LIN {X 0,Y 530.411,Z 557.197,A -85,B 0,C 180,E1 -4412.28,E2 -4412.28} C_VEL
LIN {X 0,Y 530.457,Z 555.807,A -85,B 0,C 180,E1 -4413.039,E2 -4413.039} C_VEL
LIN {X 0,Y 530.523,Z 552.892,A -85,B 0,C 180,E1 -4414.18,E2 -4414.18} C_VEL
LIN {X 0,Y 530.525,Z 548.944,A -85,B 0,C 180,E1 -4415.322,E2 -4415.322} C_VEL
LIN {X 0,Y 530.6,Z 543.257,A -85,B 0,C 180,E1 -4416.583,E2 -4416.583} C_VEL
LIN {X 0,Y 530.76,Z 536.229,A -85,B 0,C 180,E1 -4417.802,E2 -4417.802} C_VEL
LIN {X 0,Y 530.931,Z 527.981,A -85,B 0,C 180,E1 -4418.949,E2 -4418.949} C_VEL
LIN {X 0,Y 531.115,Z 519.526,A -85,B 0,C 180,E1 -4419.907,E2 -4419.907} C_VEL
LIN {X 0,Y 531.409,Z 509.082,A -85,B 0,C 180,E1 -4420.864,E2 -4420.864} C_VEL
LIN {X 0,Y 531.637,Z 497.329,A -85,B 0,C 180,E1 -4421.727,E2 -4421.727} C_VEL
LIN {X 0,Y 531.907,Z 485.461,A -85,B 0,C 180,E1 -4422.4,E2 -4422.4} C_VEL
LIN {X 0,Y 532.137,Z 473.137,A -85,B 0,C 180,E1 -4422.927,E2 -4422.927} C_VEL
LIN {X 0,Y 532.213,Z 460.93,A -85,B 0,C 180,E1 -4423.302,E2 -4423.302} C_VEL
LIN {X 0,Y 530.699,Z 451.526,A -85,B 0,C 180,E1 -4423.548,E2 -4423.548} C_VEL
LIN {X 0,Y 530.818,Z 442.755,A -85,B 0,C 180,E1 -4426.144,E2 -4426.144} C_VEL
LIN {X 0,Y 530.965,Z 433.488,A -85,B 0,C 180,E1 -4428.924,E2 -4428.924} C_VEL
LIN {X 0,Y 531.119,Z 424.221,A -85,B 0,C 180,E1 -4431.748,E2 -4431.748} C_VEL
LIN {X 0,Y 531.323,Z 414.954,A -85,B 0,C 180,E1 -4434.625,E2 -4434.625} C_VEL
LIN {X 0,Y 531.497,Z 405.493,A -85,B 0,C 180,E1 -4437.632,E2 -4437.632} C_VEL
LIN {X 0,Y 531.75,Z 395.795,A -85,B 0,C 180,E1 -4440.785,E2 -4440.785} C_VEL
LIN {X 0,Y 532.017,Z 386.981,A -85,B 0,C 180,E1 -4443.7,E2 -4443.7} C_VEL
LIN {X 0,Y 532.015,Z 380.521,A -85,B 0,C 180,E1 -4445.908,E2 -4445.908} C_VEL
LIN {X 0,Y 530.969,Z 374.349,A -85,B 0,C 180,E1 -4448.289,E2 -4448.289} C_VEL
LIN {X 0,Y 530.999,Z 374.345,A -85,B 0,C 180,E1 -4451.436,E2 -4451.436} C_VEL
LIN {X 0,Y 530.978,Z 374.348,A -85,B 0,C 180,E1 -4454.549,E2 -4454.549} C_VEL
LIN {X 0,Y 530.987,Z 374.346,A -85,B 0,C 180,E1 -4457.835,E2 -4457.835} C_VEL
LIN {X 0,Y 530.99,Z 374.345,A -85,B 0,C 180,E1 -4460.557,E2 -4460.557} C_VEL
LIN {X 0,Y 530.96,Z 374.348,A -85,B 0,C 180,E1 -4463.442,E2 -4463.442} C_VEL
LIN {X 0,Y 530.961,Z 374.348,A -85,B 0,C 180,E1 -4466.225,E2 -4466.225} C_VEL
LIN {X 0,Y 530.979,Z 374.345,A -85,B 0,C 180,E1 -4469.355,E2 -4469.355} C_VEL
LIN {X 0,Y 531.016,Z 374.342,A -85,B 0,C 180,E1 -4472.468,E2 -4472.468} C_VEL
LIN {X 0,Y 531.009,Z 374.343,A -85,B 0,C 180,E1 -4474.942,E2 -4474.942} C_VEL
LIN {X 0,Y 530.976,Z 374.348,A -85,B 0,C 180,E1 -4478.247,E2 -4478.247} C_VEL
LIN {X 0,Y 531,Z 374.344,A -85,B 0,C 180,E1 -4480.677,E2 -4480.677} C_VEL
LIN {X 0,Y 530.99,Z 374.344,A -85,B 0,C 180,E1 -4483.071,E2 -4483.071} C_VEL
LIN {X 0,Y 531.024,Z 374.341,A -85,B 0,C 180,E1 -4485.436,E2 -4485.436} C_VEL
LIN {X 0,Y 531.041,Z 374.34,A -85,B 0,C 180,E1 -4488.55,E2 -4488.55} C_VEL
LIN {X 0,Y 531.061,Z 374.335,A -85,B 0,C 180,E1 -4491.629,E2 -4491.629} C_VEL
LIN {X 0,Y 531.122,Z 374.329,A -85,B 0,C 180,E1 -4494.685,E2 -4494.685} C_VEL
LIN {X 0,Y 531.143,Z 374.326,A -85,B 0,C 180,E1 -4497.725,E2 -4497.725} C_VEL
LIN {X 0,Y 531.154,Z 374.324,A -85,B 0,C 180,E1 -4500.758,E2 -4500.758} C_VEL
LIN {X 0,Y 531.108,Z 374.33,A -85,B 0,C 180,E1 -4503.034,E2 -4503.034} C_VEL
LIN {X 0,Y 531.08,Z 374.334,A -85,B 0,C 180,E1 -4506.077,E2 -4506.077} C_VEL
LIN {X 0,Y 531.06,Z 374.337,A -85,B 0,C 180,E1 -4508.37,E2 -4508.37} C_VEL
LIN {X 0,Y 531.055,Z 374.338,A -85,B 0,C 180,E1 -4511.672,E2 -4511.672} C_VEL
LIN {X 0,Y 531.035,Z 374.338,A -85,B 0,C 180,E1 -4514.956,E2 -4514.956} C_VEL
LIN {X 0,Y 531.021,Z 374.343,A -85,B 0,C 180,E1 -4517.722,E2 -4517.722} C_VEL
LIN {X 0,Y 531.029,Z 374.34,A -85,B 0,C 180,E1 -4520.127,E2 -4520.127} C_VEL
LIN {X 0,Y 530.95,Z 374.349,A -85,B 0,C 180,E1 -4522.573,E2 -4522.573} C_VEL
LIN {X 0,Y 531.009,Z 374.344,A -85,B 0,C 180,E1 -4525.057,E2 -4525.057} C_VEL
LIN {X 0,Y 531.02,Z 374.341,A -85,B 0,C 180,E1 -4527.595,E2 -4527.595} C_VEL
LIN {X 0,Y 530.978,Z 374.345,A -85,B 0,C 180,E1 -4530.645,E2 -4530.645} C_VEL
LIN {X 0,Y 530.991,Z 374.344,A -85,B 0,C 180,E1 -4533.773,E2 -4533.773} C_VEL
LIN {X 0,Y 530.959,Z 374.349,A -85,B 0,C 180,E1 -4536.558,E2 -4536.558} C_VEL
LIN {X 0,Y 530.989,Z 374.347,A -85,B 0,C 180,E1 -4539.443,E2 -4539.443} C_VEL
LIN {X 0,Y 530.982,Z 374.346,A -85,B 0,C 180,E1 -4542.456,E2 -4542.456} C_VEL
LIN {X 0,Y 530.956,Z 374.35,A -85,B 0,C 180,E1 -4543.565,E2 -4543.565} C_VEL
LIN {X 0,Y 530.283,Z 374.432,A -85,B 0,C 180,E1 -4544.199,E2 -4544.199} C_VEL
LIN {X 0,Y 527.435,Z 374.788,A -85,B 0,C 180,E1 -4545.227,E2 -4545.227} C_VEL
LIN {X 0,Y 525.034,Z 375.089,A -85,B 0,C 180,E1 -4546.056,E2 -4546.056} C_VEL
LIN {X 0,Y 524.004,Z 375.217,A -85,B 0,C 180,E1 -4546.695,E2 -4546.695} C_VEL
LIN {X 0,Y 523.92,Z 375.226,A -85,B 0,C 180,E1 -4546.912,E2 -4546.912} C_VEL
LIN {X 0,Y 523.954,Z 375.221,A -85,B 0,C 180,E1 -4549.92,E2 -4549.92} C_VEL
LIN {X 0,Y 523.912,Z 375.228,A -85,B 0,C 180,E1 -4552.867,E2 -4552.867} C_VEL
LIN {X 0,Y 523.938,Z 375.223,A -85,B 0,C 180,E1 -4555.709,E2 -4555.709} C_VEL
LIN {X 0,Y 523.925,Z 375.225,A -85,B 0,C 180,E1 -4558.455,E2 -4558.455} C_VEL
LIN {X 0,Y 523.94,Z 375.225,A -85,B 0,C 180,E1 -4561.124,E2 -4561.124} C_VEL
LIN {X 0,Y 523.99,Z 375.215,A -85,B 0,C 180,E1 -4563.98,E2 -4563.98} C_VEL
LIN {X 0,Y 523.931,Z 375.224,A -85,B 0,C 180,E1 -4566.269,E2 -4566.269} C_VEL
LIN {X 0,Y 523.952,Z 375.222,A -85,B 0,C 180,E1 -4568.766,E2 -4568.766} C_VEL
LIN {X 0,Y 523.955,Z 375.221,A -85,B 0,C 180,E1 -4571.22,E2 -4571.22} C_VEL
LIN {X 0,Y 523.938,Z 375.223,A -85,B 0,C 180,E1 -4573.638,E2 -4573.638} C_VEL
LIN {X 0,Y 523.941,Z 375.223,A -85,B 0,C 180,E1 -4576.027,E2 -4576.027} C_VEL
LIN {X 0,Y 523.92,Z 375.227,A -85,B 0,C 180,E1 -4578.391,E2 -4578.391} C_VEL
LIN {X 0,Y 523.648,Z 375.261,A -85,B 0,C 180,E1 -4579.951,E2 -4579.951} C_VEL
LIN {X 0,Y 523.624,Z 377.586,A -85,B 0,C 180,E1 -4582.285,E2 -4582.285} C_VEL
LIN {X 0,Y 523.616,Z 381.014,A -85,B 0,C 180,E1 -4585.379,E2 -4585.379} C_VEL
LIN {X 0,Y 523.462,Z 384.449,A -85,B 0,C 180,E1 -4588.46,E2 -4588.46} C_VEL
LIN {X 0,Y 523.412,Z 386.99,A -85,B 0,C 180,E1 -4590.768,E2 -4590.768} C_VEL
LIN {X 0,Y 523.525,Z 390.404,A -85,B 0,C 180,E1 -4593.847,E2 -4593.847} C_VEL
LIN {X 0,Y 523.463,Z 393.361,A -85,B 0,C 180,E1 -4596.525,E2 -4596.525} C_VEL
LIN {X 0,Y 523.359,Z 396.588,A -85,B 0,C 180,E1 -4599.393,E2 -4599.393} C_VEL
LIN {X 0,Y 525.379,Z 407.996,A -85,B 0,C 180,E1 -4599.746,E2 -4599.746} C_VEL
LIN {X 0,Y 525.184,Z 420.456,A -85,B 0,C 180,E1 -4600.211,E2 -4600.211} C_VEL
LIN {X 0,Y 524.864,Z 432.201,A -85,B 0,C 180,E1 -4600.803,E2 -4600.803} C_VEL
LIN {X 0,Y 524.583,Z 444.103,A -85,B 0,C 180,E1 -4601.591,E2 -4601.591} C_VEL
LIN {X 0,Y 524.273,Z 454.764,A -85,B 0,C 180,E1 -4602.482,E2 -4602.482} C_VEL
LIN {X 0,Y 524.031,Z 463.464,A -85,B 0,C 180,E1 -4603.375,E2 -4603.375} C_VEL
LIN {X 0,Y 523.843,Z 471.463,A -85,B 0,C 180,E1 -4604.369,E2 -4604.369} C_VEL
LIN {X 0,Y 523.652,Z 479.258,A -85,B 0,C 180,E1 -4605.569,E2 -4605.569} C_VEL
LIN {X 0,Y 523.518,Z 485.51,A -85,B 0,C 180,E1 -4606.774,E2 -4606.774} C_VEL
LIN {X 0,Y 523.41,Z 490.453,A -85,B 0,C 180,E1 -4607.987,E2 -4607.987} C_VEL
LIN {X 0,Y 523.368,Z 494.214,A -85,B 0,C 180,E1 -4609.206,E2 -4609.206} C_VEL
LIN {X 0,Y 523.267,Z 496.898,A -85,B 0,C 180,E1 -4610.437,E2 -4610.437} C_VEL
LIN {X 0,Y 523.271,Z 498.106,A -85,B 0,C 180,E1 -4611.26,E2 -4611.26} C_VEL
LIN {X 0,Y 523.292,Z 498.835,A -85,B 0,C 180,E1 -4612.087,E2 -4612.087} C_VEL
LIN {X 0,Y 523.268,Z 499.146,A -85,B 0,C 180,E1 -4612.921,E2 -4612.921} C_VEL
LIN {X 0,Y 523.296,Z 498.812,A -85,B 0,C 180,E1 -4614.04,E2 -4614.04} C_VEL
LIN {X 0,Y 523.299,Z 497.244,A -85,B 0,C 180,E1 -4615.451,E2 -4615.451} C_VEL
LIN {X 0,Y 523.354,Z 494.625,A -85,B 0,C 180,E1 -4616.733,E2 -4616.733} C_VEL
LIN {X 0,Y 523.41,Z 490.733,A -85,B 0,C 180,E1 -4618.029,E2 -4618.029} C_VEL
LIN {X 0,Y 523.542,Z 484.799,A -85,B 0,C 180,E1 -4619.473,E2 -4619.473} C_VEL
LIN {X 0,Y 523.685,Z 478.485,A -85,B 0,C 180,E1 -4620.659,E2 -4620.659} C_VEL
LIN {X 0,Y 523.858,Z 471.102,A -85,B 0,C 180,E1 -4621.772,E2 -4621.772} C_VEL
LIN {X 0,Y 524.127,Z 461.895,A -85,B 0,C 180,E1 -4622.89,E2 -4622.89} C_VEL
LIN {X 0,Y 524.363,Z 452.696,A -85,B 0,C 180,E1 -4623.8,E2 -4623.8} C_VEL
LIN {X 0,Y 524.619,Z 443,A -85,B 0,C 180,E1 -4624.585,E2 -4624.585} C_VEL
LIN {X 0,Y 524.919,Z 430.95,A -85,B 0,C 180,E1 -4625.358,E2 -4625.358} C_VEL
LIN {X 0,Y 525.195,Z 419.142,A -85,B 0,C 180,E1 -4625.939,E2 -4625.939} C_VEL
LIN {X 0,Y 525.253,Z 406.72,A -85,B 0,C 180,E1 -4626.391,E2 -4626.391} C_VEL
LIN {X 0,Y 523.353,Z 396.648,A -85,B 0,C 180,E1 -4626.718,E2 -4626.718} C_VEL
LIN {X 0,Y 523.384,Z 392.89,A -85,B 0,C 180,E1 -4630.129,E2 -4630.129} C_VEL
LIN {X 0,Y 523.465,Z 389.19,A -85,B 0,C 180,E1 -4633.531,E2 -4633.531} C_VEL
LIN {X 0,Y 523.499,Z 385.993,A -85,B 0,C 180,E1 -4636.461,E2 -4636.461} C_VEL
LIN {X 0,Y 523.559,Z 383.372,A -85,B 0,C 180,E1 -4638.871,E2 -4638.871} C_VEL
LIN {X 0,Y 523.579,Z 379.53,A -85,B 0,C 180,E1 -4642.365,E2 -4642.365} C_VEL
LIN {X 0,Y 523.642,Z 376.712,A -85,B 0,C 180,E1 -4644.951,E2 -4644.951} C_VEL
LIN {X 0,Y 523.652,Z 375.261,A -85,B 0,C 180,E1 -4646.312,E2 -4646.312} C_VEL
LIN {X 0,Y 523.863,Z 375.235,A -85,B 0,C 180,E1 -4648.452,E2 -4648.452} C_VEL
LIN {X 0,Y 523.933,Z 375.225,A -85,B 0,C 180,E1 -4651.125,E2 -4651.125} C_VEL
LIN {X 0,Y 523.967,Z 375.22,A -85,B 0,C 180,E1 -4653.979,E2 -4653.979} C_VEL
LIN {X 0,Y 523.943,Z 375.224,A -85,B 0,C 180,E1 -4656.271,E2 -4656.271} C_VEL
LIN {X 0,Y 523.94,Z 375.222,A -85,B 0,C 180,E1 -4658.766,E2 -4658.766} C_VEL
LIN {X 0,Y 523.936,Z 375.221,A -85,B 0,C 180,E1 -4661.22,E2 -4661.22} C_VEL
LIN {X 0,Y 523.92,Z 375.223,A -85,B 0,C 180,E1 -4663.638,E2 -4663.638} C_VEL
LIN {X 0,Y 523.923,Z 375.225,A -85,B 0,C 180,E1 -4666.028,E2 -4666.028} C_VEL
LIN {X 0,Y 523.99,Z 375.217,A -85,B 0,C 180,E1 -4668.394,E2 -4668.394} C_VEL
LIN {X 0,Y 523.989,Z 375.217,A -85,B 0,C 180,E1 -4671.516,E2 -4671.516} C_VEL
LIN {X 0,Y 524.086,Z 375.203,A -85,B 0,C 180,E1 -4674.614,E2 -4674.614} C_VEL
LIN {X 0,Y 524.098,Z 375.202,A -85,B 0,C 180,E1 -4677.694,E2 -4677.694} C_VEL
LIN {X 0,Y 524.108,Z 375.204,A -85,B 0,C 180,E1 -4680.768,E2 -4680.768} C_VEL
LIN {X 0,Y 524.06,Z 375.207,A -85,B 0,C 180,E1 -4683.075,E2 -4683.075} C_VEL
LIN {X 0,Y 524.027,Z 375.214,A -85,B 0,C 180,E1 -4686.159,E2 -4686.159} C_VEL
LIN {X 0,Y 523.982,Z 375.216,A -85,B 0,C 180,E1 -4689.262,E2 -4689.262} C_VEL
LIN {X 0,Y 524.003,Z 375.215,A -85,B 0,C 180,E1 -4691.752,E2 -4691.752} C_VEL
LIN {X 0,Y 523.972,Z 375.217,A -85,B 0,C 180,E1 -4695.053,E2 -4695.053} C_VEL
LIN {X 0,Y 523.945,Z 375.221,A -85,B 0,C 180,E1 -4697.97,E2 -4697.97} C_VEL
LIN {X 0,Y 523.955,Z 375.219,A -85,B 0,C 180,E1 -4700.411,E2 -4700.411} C_VEL
LIN {X 0,Y 523.942,Z 375.222,A -85,B 0,C 180,E1 -4702.892,E2 -4702.892} C_VEL
LIN {X 0,Y 523.938,Z 375.223,A -85,B 0,C 180,E1 -4705.42,E2 -4705.42} C_VEL
LIN {X 0,Y 523.953,Z 375.223,A -85,B 0,C 180,E1 -4708,E2 -4708} C_VEL
LIN {X 0,Y 523.93,Z 375.224,A -85,B 0,C 180,E1 -4710.857,E2 -4710.857} C_VEL
LIN {X 0,Y 523.945,Z 375.221,A -85,B 0,C 180,E1 -4713.736,E2 -4713.736} C_VEL
LIN {X 0,Y 523.91,Z 375.225,A -85,B 0,C 180,E1 -4716.406,E2 -4716.406} C_VEL
LIN {X 0,Y 523.915,Z 375.225,A -85,B 0,C 180,E1 -4719.085,E2 -4719.085} C_VEL
LIN {X 0,Y 523.951,Z 375.222,A -85,B 0,C 180,E1 -4722.119,E2 -4722.119} C_VEL
LIN {X 0,Y 523.943,Z 375.227,A -85,B 0,C 180,E1 -4725.31,E2 -4725.31} C_VEL
LIN {X 0,Y 523.963,Z 375.221,A -85,B 0,C 180,E1 -4728.689,E2 -4728.689} C_VEL
LIN {X 0,Y 523.937,Z 375.408,A -85,B 0,C 180,E1 -4731.536,E2 -4731.536} C_VEL
LIN {X 0,Y 525.033,Z 381.484,A -85,B 0,C 180,E1 -4733.918,E2 -4733.918} C_VEL
LIN {X 0,Y 525.046,Z 387.672,A -85,B 0,C 180,E1 -4736.089,E2 -4736.089} C_VEL
LIN {X 0,Y 524.764,Z 396.482,A -85,B 0,C 180,E1 -4738.996,E2 -4738.996} C_VEL
LIN {X 0,Y 524.531,Z 406.097,A -85,B 0,C 180,E1 -4742.167,E2 -4742.167} C_VEL
LIN {X 0,Y 524.307,Z 414.964,A -85,B 0,C 180,E1 -4745.026,E2 -4745.026} C_VEL
LIN {X 0,Y 524.12,Z 424.231,A -85,B 0,C 180,E1 -4747.95,E2 -4747.95} C_VEL
LIN {X 0,Y 523.924,Z 433.498,A -85,B 0,C 180,E1 -4750.815,E2 -4750.815} C_VEL
LIN {X 0,Y 523.761,Z 442.766,A -85,B 0,C 180,E1 -4753.635,E2 -4753.635} C_VEL
LIN {X 0,Y 523.637,Z 451.536,A -85,B 0,C 180,E1 -4756.269,E2 -4756.269} C_VEL
LIN {X 0,Y 525.451,Z 463.334,A -85,B 0,C 180,E1 -4756.588,E2 -4756.588} C_VEL
LIN {X 0,Y 525.22,Z 475.817,A -85,B 0,C 180,E1 -4757.001,E2 -4757.001} C_VEL
LIN {X 0,Y 524.933,Z 487.442,A -85,B 0,C 180,E1 -4757.534,E2 -4757.534} C_VEL
LIN {X 0,Y 524.658,Z 498.85,A -85,B 0,C 180,E1 -4758.219,E2 -4758.219} C_VEL
LIN {X 0,Y 524.388,Z 510.282,A -85,B 0,C 180,E1 -4759.089,E2 -4759.089} C_VEL
LIN {X 0,Y 524.095,Z 519.555,A -85,B 0,C 180,E1 -4759.962,E2 -4759.962} C_VEL
LIN {X 0,Y 523.895,Z 528.004,A -85,B 0,C 180,E1 -4760.933,E2 -4760.933} C_VEL
LIN {X 0,Y 523.686,Z 536.247,A -85,B 0,C 180,E1 -4762.095,E2 -4762.095} C_VEL
LIN {X 0,Y 523.573,Z 541.877,A -85,B 0,C 180,E1 -4763.063,E2 -4763.063} C_VEL
LIN {X 0,Y 523.543,Z 547.373,A -85,B 0,C 180,E1 -4764.223,E2 -4764.223} C_VEL
LIN {X 0,Y 523.36,Z 551.682,A -85,B 0,C 180,E1 -4765.38,E2 -4765.38} C_VEL
LIN {X 0,Y 523.443,Z 553.962,A -85,B 0,C 180,E1 -4766.152,E2 -4766.152} C_VEL
LIN {X 0,Y 523.367,Z 555.811,A -85,B 0,C 180,E1 -4766.922,E2 -4766.922} C_VEL
LIN {X 0,Y 523.335,Z 557.199,A -85,B 0,C 180,E1 -4767.693,E2 -4767.693} C_VEL
LIN {X 0,Y 523.25,Z 558.786,A -85,B 0,C 180,E1 -4769.232,E2 -4769.232} C_VEL
LIN {X 0,Y 523.246,Z 559,A -85,B 0,C 180,E1 -4770.001,E2 -4770.001} C_VEL
LIN {X 0,Y 523.275,Z 558.184,A -85,B 0,C 180,E1 -4771.541,E2 -4771.541} C_VEL
LIN {X 0,Y 523.335,Z 557.197,A -85,B 0,C 180,E1 -4772.31,E2 -4772.31} C_VEL
LIN {X 0,Y 523.368,Z 555.807,A -85,B 0,C 180,E1 -4773.08,E2 -4773.08} C_VEL
LIN {X 0,Y 523.442,Z 552.892,A -85,B 0,C 180,E1 -4774.236,E2 -4774.236} C_VEL
LIN {X 0,Y 523.464,Z 548.944,A -85,B 0,C 180,E1 -4775.394,E2 -4775.394} C_VEL
LIN {X 0,Y 523.525,Z 543.72,A -85,B 0,C 180,E1 -4776.582,E2 -4776.582} C_VEL
LIN {X 0,Y 523.666,Z 537.46,A -85,B 0,C 180,E1 -4777.714,E2 -4777.714} C_VEL
LIN {X 0,Y 523.856,Z 529.468,A -85,B 0,C 180,E1 -4778.877,E2 -4778.877} C_VEL
LIN {X 0,Y 524.087,Z 521.323,A -85,B 0,C 180,E1 -4779.846,E2 -4779.846} C_VEL
LIN {X 0,Y 524.352,Z 511.386,A -85,B 0,C 180,E1 -4780.817,E2 -4780.817} C_VEL
LIN {X 0,Y 524.652,Z 500.233,A -85,B 0,C 180,E1 -4781.686,E2 -4781.686} C_VEL
LIN {X 0,Y 524.894,Z 489.153,A -85,B 0,C 180,E1 -4782.372,E2 -4782.372} C_VEL
LIN {X 0,Y 525.187,Z 476.95,A -85,B 0,C 180,E1 -4782.954,E2 -4782.954} C_VEL
LIN {X 0,Y 525.384,Z 464.13,A -85,B 0,C 180,E1 -4783.392,E2 -4783.392} C_VEL
LIN {X 0,Y 524.753,Z 458.309,A -85,B 0,C 180,E1 -4783.556,E2 -4783.556} C_VEL
LIN {X 0,Y 523.638,Z 451.526,A -85,B 0,C 180,E1 -4783.734,E2 -4783.734} C_VEL
LIN {X 0,Y 523.766,Z 442.755,A -85,B 0,C 180,E1 -4786.368,E2 -4786.368} C_VEL
LIN {X 0,Y 523.931,Z 433.488,A -85,B 0,C 180,E1 -4789.188,E2 -4789.188} C_VEL
LIN {X 0,Y 524.13,Z 423.437,A -85,B 0,C 180,E1 -4792.299,E2 -4792.299} C_VEL
LIN {X 0,Y 524.354,Z 413.63,A -85,B 0,C 180,E1 -4795.399,E2 -4795.399} C_VEL
LIN {X 0,Y 524.605,Z 404.363,A -85,B 0,C 180,E1 -4798.398,E2 -4798.398} C_VEL
LIN {X 0,Y 524.823,Z 394.974,A -85,B 0,C 180,E1 -4801.485,E2 -4801.485} C_VEL
LIN {X 0,Y 525.085,Z 386.898,A -85,B 0,C 180,E1 -4804.206,E2 -4804.206} C_VEL
LIN {X 0,Y 525.016,Z 381.504,A -85,B 0,C 180,E1 -4806.087,E2 -4806.087} C_VEL
LIN {X 0,Y 523.939,Z 375.225,A -85,B 0,C 180,E1 -4808.591,E2 -4808.591} C_VEL
LIN {X 0,Y 523.962,Z 375.222,A -85,B 0,C 180,E1 -4811.311,E2 -4811.311} C_VEL
LIN {X 0,Y 523.947,Z 375.223,A -85,B 0,C 180,E1 -4814.69,E2 -4814.69} C_VEL
LIN {X 0,Y 523.957,Z 375.221,A -85,B 0,C 180,E1 -4817.881,E2 -4817.881} C_VEL
LIN {X 0,Y 523.924,Z 375.226,A -85,B 0,C 180,E1 -4820.915,E2 -4820.915} C_VEL
LIN {X 0,Y 523.905,Z 375.227,A -85,B 0,C 180,E1 -4823.825,E2 -4823.825} C_VEL
LIN {X 0,Y 523.918,Z 375.226,A -85,B 0,C 180,E1 -4826.634,E2 -4826.634} C_VEL
LIN {X 0,Y 523.961,Z 375.219,A -85,B 0,C 180,E1 -4829.356,E2 -4829.356} C_VEL
LIN {X 0,Y 523.981,Z 375.219,A -85,B 0,C 180,E1 -4832.282,E2 -4832.282} C_VEL
LIN {X 0,Y 523.957,Z 375.221,A -85,B 0,C 180,E1 -4834.581,E2 -4834.581} C_VEL
LIN {X 0,Y 523.915,Z 375.227,A -85,B 0,C 180,E1 -4837.107,E2 -4837.107} C_VEL
LIN {X 0,Y 523.984,Z 375.217,A -85,B 0,C 180,E1 -4839.866,E2 -4839.866} C_VEL
LIN {X 0,Y 523.971,Z 375.219,A -85,B 0,C 180,E1 -4842.837,E2 -4842.837} C_VEL
LIN {X 0,Y 523.981,Z 375.217,A -85,B 0,C 180,E1 -4845.236,E2 -4845.236} C_VEL
LIN {X 0,Y 524.017,Z 375.214,A -85,B 0,C 180,E1 -4848.394,E2 -4848.394} C_VEL
LIN {X 0,Y 524.009,Z 375.213,A -85,B 0,C 180,E1 -4851.516,E2 -4851.516} C_VEL
LIN {X 0,Y 524.084,Z 375.206,A -85,B 0,C 180,E1 -4854.614,E2 -4854.614} C_VEL
LIN {X 0,Y 524.115,Z 375.201,A -85,B 0,C 180,E1 -4857.694,E2 -4857.694} C_VEL
LIN {X 0,Y 524.125,Z 375.2,A -85,B 0,C 180,E1 -4860.768,E2 -4860.768} C_VEL
LIN {X 0,Y 524.075,Z 375.206,A -85,B 0,C 180,E1 -4863.075,E2 -4863.075} C_VEL
LIN {X 0,Y 524.041,Z 375.212,A -85,B 0,C 180,E1 -4866.159,E2 -4866.159} C_VEL
LIN {X 0,Y 524.009,Z 375.214,A -85,B 0,C 180,E1 -4868.484,E2 -4868.484} C_VEL
LIN {X 0,Y 524.007,Z 375.215,A -85,B 0,C 180,E1 -4871.739,E2 -4871.739} C_VEL
LIN {X 0,Y 523.997,Z 375.215,A -85,B 0,C 180,E1 -4875.052,E2 -4875.052} C_VEL
LIN {X 0,Y 523.967,Z 375.22,A -85,B 0,C 180,E1 -4877.969,E2 -4877.969} C_VEL
LIN {X 0,Y 523.976,Z 375.218,A -85,B 0,C 180,E1 -4880.41,E2 -4880.41} C_VEL
LIN {X 0,Y 523.915,Z 375.226,A -85,B 0,C 180,E1 -4882.893,E2 -4882.893} C_VEL
LIN {X 0,Y 523.956,Z 375.221,A -85,B 0,C 180,E1 -4885.418,E2 -4885.418} C_VEL
LIN {X 0,Y 523.974,Z 375.22,A -85,B 0,C 180,E1 -4887.999,E2 -4887.999} C_VEL
LIN {X 0,Y 523.949,Z 375.221,A -85,B 0,C 180,E1 -4890.854,E2 -4890.854} C_VEL
LIN {X 0,Y 523.963,Z 375.22,A -85,B 0,C 180,E1 -4893.734,E2 -4893.734} C_VEL
LIN {X 0,Y 523.907,Z 375.227,A -85,B 0,C 180,E1 -4896.401,E2 -4896.401} C_VEL
LIN {X 0,Y 523.923,Z 375.225,A -85,B 0,C 180,E1 -4899.085,E2 -4899.085} C_VEL
LIN {X 0,Y 523.956,Z 375.22,A -85,B 0,C 180,E1 -4902.119,E2 -4902.119} C_VEL
LIN {X 0,Y 523.947,Z 375.222,A -85,B 0,C 180,E1 -4905.31,E2 -4905.31} C_VEL
LIN {X 0,Y 523.92,Z 375.226,A -85,B 0,C 180,E1 -4906.912,E2 -4906.912} C_VEL
LIN {X 0,Y 523.257,Z 375.309,A -85,B 0,C 180,E1 -4907.554,E2 -4907.554} C_VEL
LIN {X 0,Y 520.416,Z 375.661,A -85,B 0,C 180,E1 -4908.595,E2 -4908.595} C_VEL
LIN {X 0,Y 518.011,Z 375.962,A -85,B 0,C 180,E1 -4909.434,E2 -4909.434} C_VEL
LIN {X 0,Y 516.974,Z 376.09,A -85,B 0,C 180,E1 -4910.082,E2 -4910.082} C_VEL
LIN {X 0,Y 516.887,Z 376.1,A -85,B 0,C 180,E1 -4910.301,E2 -4910.301} C_VEL
LIN {X 0,Y 516.882,Z 376.102,A -85,B 0,C 180,E1 -4913.342,E2 -4913.342} C_VEL
